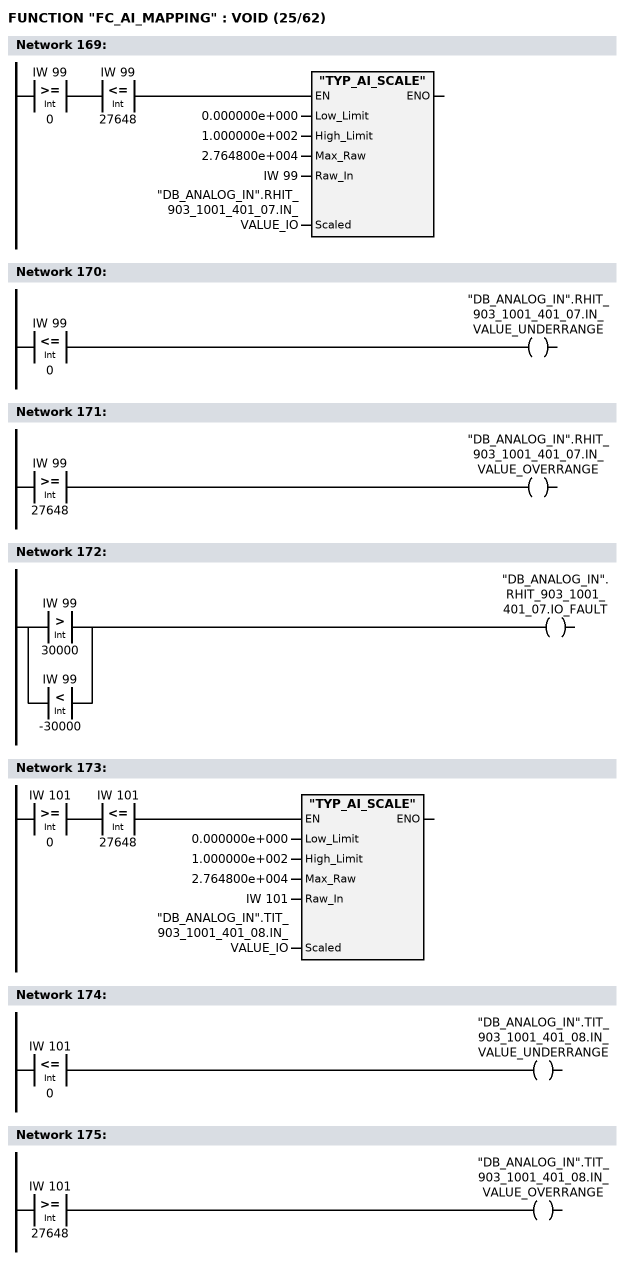

      A(    ;
      L     IW      99;
      L     0;
      >=I   ;
      )     ;
      A(    ;
      L     IW      99;

      L     27648;
      <=I   ;
      )     ;
      JNB   _02b;
      CALL "TYP_AI_SCALE" (
           Low_Limit                := 0.000000e+000,
           High_Limit               := 1.000000e+002,
           Max_Raw                  := 2.764800e+004,
           Raw_In                   := IW      99,
           Scaled                   := "DB_ANALOG_IN".RHIT_903_1001_401_07.IN_VALUE_IO);
_02b: NOP   0;
NETWORK
TITLE =

      L     IW      99;
      L     0;
      <=I   ;
      =     "DB_ANALOG_IN".RHIT_903_1001_401_07.IN_VALUE_UNDERRANGE;
NETWORK
TITLE =

      L     IW      99;
      L     27648;
      >=I   ;
      =     "DB_ANALOG_IN".RHIT_903_1001_401_07.IN_VALUE_OVERRANGE;
NETWORK
TITLE =

      O(    ;
      L     IW      99;
      L     30000;
      >I    ;
      )     ;
      O(    ;
      L     IW      99;
      L     -30000;
      <I    ;
      )     ;
      =     "DB_ANALOG_IN".RHIT_903_1001_401_07.IO_FAULT;

NETWORK
TITLE =

      A(    ;
      L     IW      101;
      L     0;
      >=I   ;
      )     ;
      A(    ;
      L     IW      101;

      L     27648;
      <=I   ;
      )     ;
      JNB   _02c;
      CALL "TYP_AI_SCALE" (
           Low_Limit                := 0.000000e+000,
           High_Limit               := 1.000000e+002,
           Max_Raw                  := 2.764800e+004,
           Raw_In                   := IW      101,
           Scaled                   := "DB_ANALOG_IN".TIT_903_1001_401_08.IN_VALUE_IO);
_02c: NOP   0;
NETWORK
TITLE =

      L     IW      101;
      L     0;
      <=I   ;
      =     "DB_ANALOG_IN".TIT_903_1001_401_08.IN_VALUE_UNDERRANGE;
NETWORK
TITLE =

      L     IW      101;
      L     27648;
      >=I   ;
      =     "DB_ANALOG_IN".TIT_903_1001_401_08.IN_VALUE_OVERRANGE;
NETWORK
TITLE =
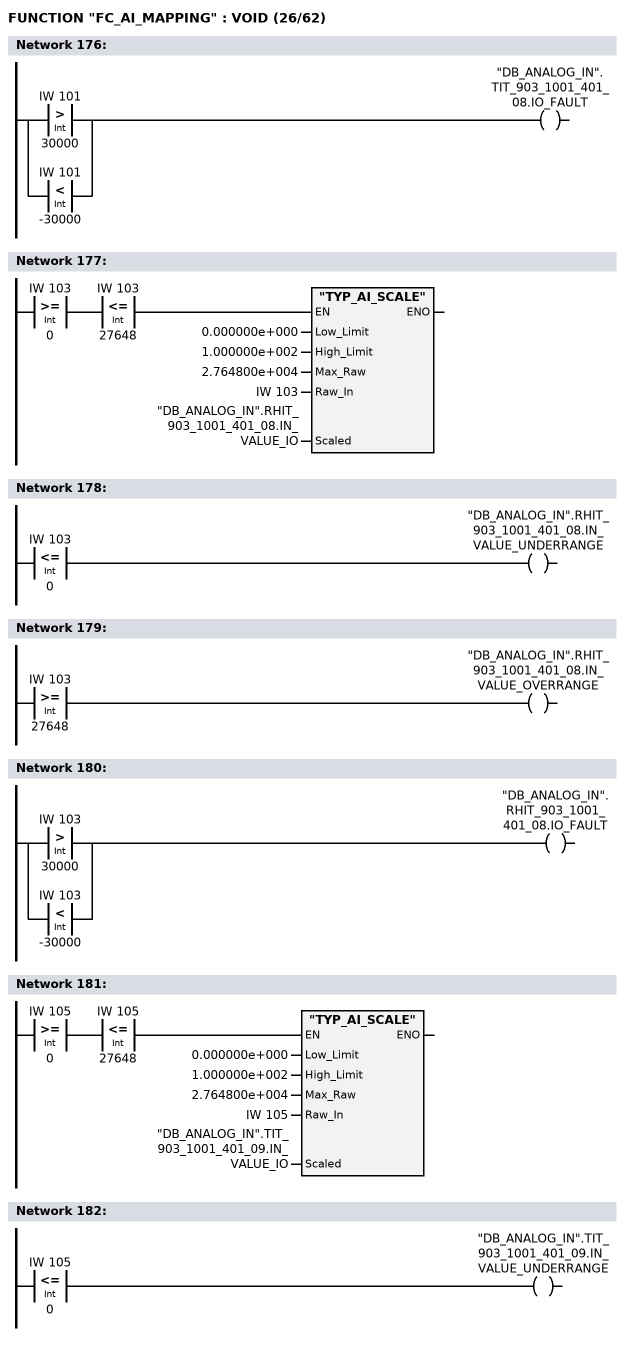

      O(    ;
      L     IW      101;
      L     30000;
      >I    ;
      )     ;
      O(    ;
      L     IW      101;
      L     -30000;
      <I    ;
      )     ;
      =     "DB_ANALOG_IN".TIT_903_1001_401_08.IO_FAULT;

NETWORK
TITLE =

      A(    ;
      L     IW      103;
      L     0;
      >=I   ;
      )     ;
      A(    ;
      L     IW      103;

      L     27648;
      <=I   ;
      )     ;
      JNB   _02d;
      CALL "TYP_AI_SCALE" (
           Low_Limit                := 0.000000e+000,
           High_Limit               := 1.000000e+002,
           Max_Raw                  := 2.764800e+004,
           Raw_In                   := IW      103,
           Scaled                   := "DB_ANALOG_IN".RHIT_903_1001_401_08.IN_VALUE_IO);
_02d: NOP   0;
NETWORK
TITLE =

      L     IW      103;
      L     0;
      <=I   ;
      =     "DB_ANALOG_IN".RHIT_903_1001_401_08.IN_VALUE_UNDERRANGE;
NETWORK
TITLE =

      L     IW      103;
      L     27648;
      >=I   ;
      =     "DB_ANALOG_IN".RHIT_903_1001_401_08.IN_VALUE_OVERRANGE;
NETWORK
TITLE =

      O(    ;
      L     IW      103;
      L     30000;
      >I    ;
      )     ;
      O(    ;
      L     IW      103;
      L     -30000;
      <I    ;
      )     ;
      =     "DB_ANALOG_IN".RHIT_903_1001_401_08.IO_FAULT;

NETWORK
TITLE =

      A(    ;
      L     IW      105;
      L     0;
      >=I   ;
      )     ;
      A(    ;
      L     IW      105;

      L     27648;
      <=I   ;
      )     ;
      JNB   _02e;
      CALL "TYP_AI_SCALE" (
           Low_Limit                := 0.000000e+000,
           High_Limit               := 1.000000e+002,
           Max_Raw                  := 2.764800e+004,
           Raw_In                   := IW      105,
           Scaled                   := "DB_ANALOG_IN".TIT_903_1001_401_09.IN_VALUE_IO);
_02e: NOP   0;
NETWORK
TITLE =

      L     IW      105;
      L     0;
      <=I   ;
      =     "DB_ANALOG_IN".TIT_903_1001_401_09.IN_VALUE_UNDERRANGE;
NETWORK
TITLE =
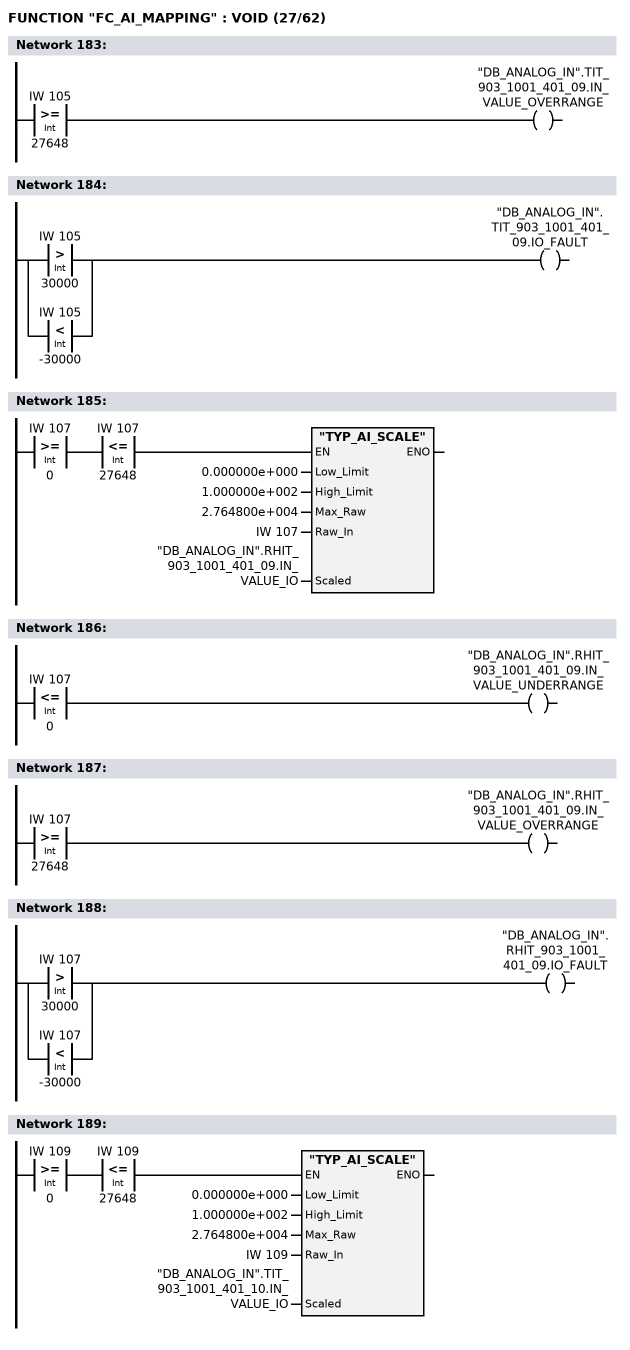

      L     IW      105;
      L     27648;
      >=I   ;
      =     "DB_ANALOG_IN".TIT_903_1001_401_09.IN_VALUE_OVERRANGE;
NETWORK
TITLE =

      O(    ;
      L     IW      105;
      L     30000;
      >I    ;
      )     ;
      O(    ;
      L     IW      105;
      L     -30000;
      <I    ;
      )     ;
      =     "DB_ANALOG_IN".TIT_903_1001_401_09.IO_FAULT;

NETWORK
TITLE =

      A(    ;
      L     IW      107;
      L     0;
      >=I   ;
      )     ;
      A(    ;
      L     IW      107;

      L     27648;
      <=I   ;
      )     ;
      JNB   _02f;
      CALL "TYP_AI_SCALE" (
           Low_Limit                := 0.000000e+000,
           High_Limit               := 1.000000e+002,
           Max_Raw                  := 2.764800e+004,
           Raw_In                   := IW      107,
           Scaled                   := "DB_ANALOG_IN".RHIT_903_1001_401_09.IN_VALUE_IO);
_02f: NOP   0;
NETWORK
TITLE =

      L     IW      107;
      L     0;
      <=I   ;
      =     "DB_ANALOG_IN".RHIT_903_1001_401_09.IN_VALUE_UNDERRANGE;
NETWORK
TITLE =

      L     IW      107;
      L     27648;
      >=I   ;
      =     "DB_ANALOG_IN".RHIT_903_1001_401_09.IN_VALUE_OVERRANGE;
NETWORK
TITLE =

      O(    ;
      L     IW      107;
      L     30000;
      >I    ;
      )     ;
      O(    ;
      L     IW      107;
      L     -30000;
      <I    ;
      )     ;
      =     "DB_ANALOG_IN".RHIT_903_1001_401_09.IO_FAULT;

NETWORK
TITLE =

      A(    ;
      L     IW      109;
      L     0;
      >=I   ;
      )     ;
      A(    ;
      L     IW      109;

      L     27648;
      <=I   ;
      )     ;
      JNB   _030;
      CALL "TYP_AI_SCALE" (
           Low_Limit                := 0.000000e+000,
           High_Limit               := 1.000000e+002,
           Max_Raw                  := 2.764800e+004,
           Raw_In                   := IW      109,
           Scaled                   := "DB_ANALOG_IN".TIT_903_1001_401_10.IN_VALUE_IO);
_030: NOP   0;
NETWORK
TITLE =
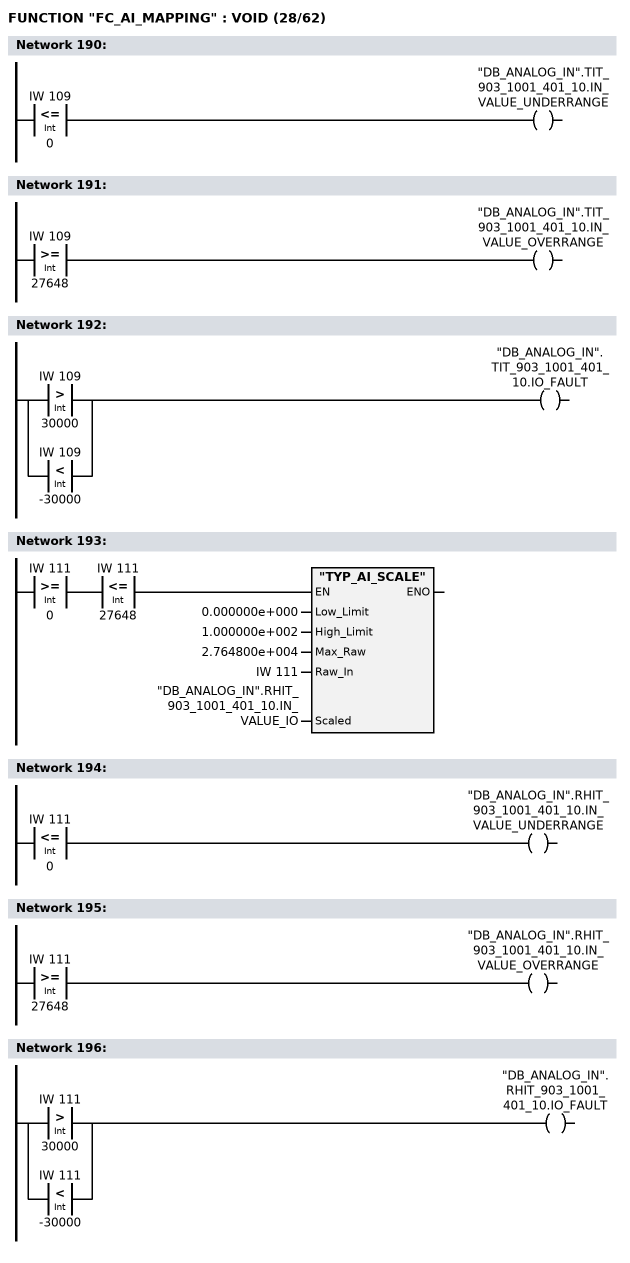

      L     IW      109;
      L     0;
      <=I   ;
      =     "DB_ANALOG_IN".TIT_903_1001_401_10.IN_VALUE_UNDERRANGE;
NETWORK
TITLE =

      L     IW      109;
      L     27648;
      >=I   ;
      =     "DB_ANALOG_IN".TIT_903_1001_401_10.IN_VALUE_OVERRANGE;
NETWORK
TITLE =

      O(    ;
      L     IW      109;
      L     30000;
      >I    ;
      )     ;
      O(    ;
      L     IW      109;
      L     -30000;
      <I    ;
      )     ;
      =     "DB_ANALOG_IN".TIT_903_1001_401_10.IO_FAULT;

NETWORK
TITLE =

      A(    ;
      L     IW      111;
      L     0;
      >=I   ;
      )     ;
      A(    ;
      L     IW      111;

      L     27648;
      <=I   ;
      )     ;
      JNB   _031;
      CALL "TYP_AI_SCALE" (
           Low_Limit                := 0.000000e+000,
           High_Limit               := 1.000000e+002,
           Max_Raw                  := 2.764800e+004,
           Raw_In                   := IW      111,
           Scaled                   := "DB_ANALOG_IN".RHIT_903_1001_401_10.IN_VALUE_IO);
_031: NOP   0;
NETWORK
TITLE =

      L     IW      111;
      L     0;
      <=I   ;
      =     "DB_ANALOG_IN".RHIT_903_1001_401_10.IN_VALUE_UNDERRANGE;
NETWORK
TITLE =

      L     IW      111;
      L     27648;
      >=I   ;
      =     "DB_ANALOG_IN".RHIT_903_1001_401_10.IN_VALUE_OVERRANGE;
NETWORK
TITLE =

      O(    ;
      L     IW      111;
      L     30000;
      >I    ;
      )     ;
      O(    ;
      L     IW      111;
      L     -30000;
      <I    ;
      )     ;
      =     "DB_ANALOG_IN".RHIT_903_1001_401_10.IO_FAULT;

NETWORK
TITLE =
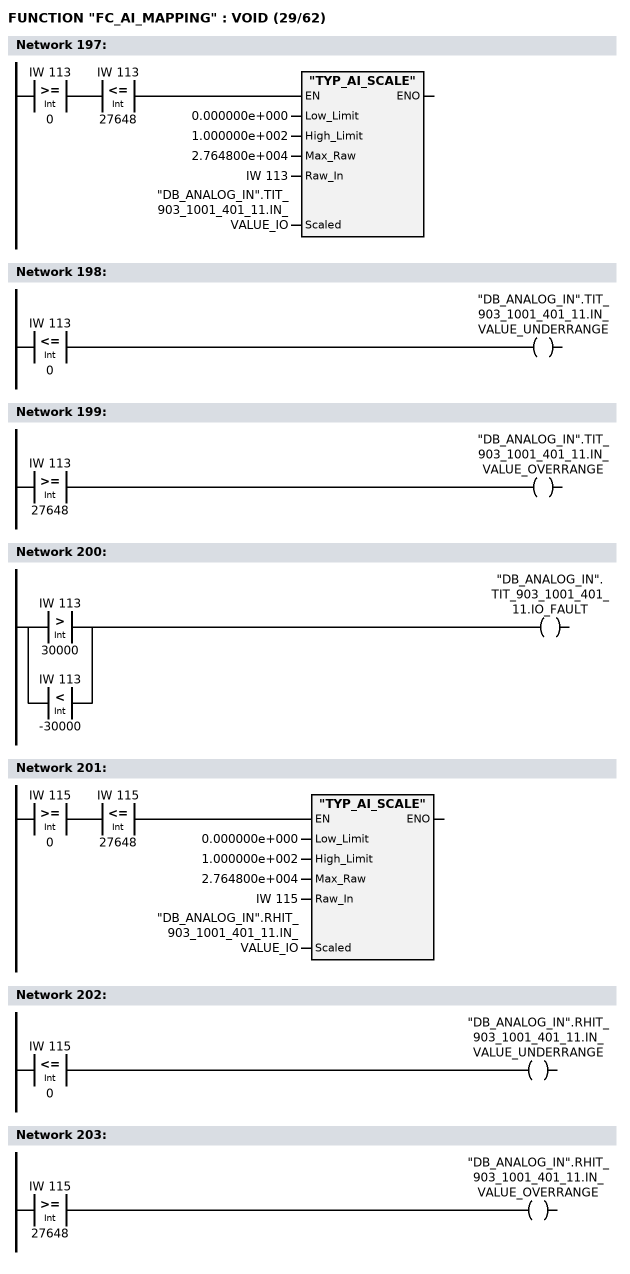

      A(    ;
      L     IW      113;
      L     0;
      >=I   ;
      )     ;
      A(    ;
      L     IW      113;

      L     27648;
      <=I   ;
      )     ;
      JNB   _032;
      CALL "TYP_AI_SCALE" (
           Low_Limit                := 0.000000e+000,
           High_Limit               := 1.000000e+002,
           Max_Raw                  := 2.764800e+004,
           Raw_In                   := IW      113,
           Scaled                   := "DB_ANALOG_IN".TIT_903_1001_401_11.IN_VALUE_IO);
_032: NOP   0;
NETWORK
TITLE =

      L     IW      113;
      L     0;
      <=I   ;
      =     "DB_ANALOG_IN".TIT_903_1001_401_11.IN_VALUE_UNDERRANGE;
NETWORK
TITLE =

      L     IW      113;
      L     27648;
      >=I   ;
      =     "DB_ANALOG_IN".TIT_903_1001_401_11.IN_VALUE_OVERRANGE;
NETWORK
TITLE =

      O(    ;
      L     IW      113;
      L     30000;
      >I    ;
      )     ;
      O(    ;
      L     IW      113;
      L     -30000;
      <I    ;
      )     ;
      =     "DB_ANALOG_IN".TIT_903_1001_401_11.IO_FAULT;

NETWORK
TITLE =

      A(    ;
      L     IW      115;
      L     0;
      >=I   ;
      )     ;
      A(    ;
      L     IW      115;

      L     27648;
      <=I   ;
      )     ;
      JNB   _033;
      CALL "TYP_AI_SCALE" (
           Low_Limit                := 0.000000e+000,
           High_Limit               := 1.000000e+002,
           Max_Raw                  := 2.764800e+004,
           Raw_In                   := IW      115,
           Scaled                   := "DB_ANALOG_IN".RHIT_903_1001_401_11.IN_VALUE_IO);
_033: NOP   0;
NETWORK
TITLE =

      L     IW      115;
      L     0;
      <=I   ;
      =     "DB_ANALOG_IN".RHIT_903_1001_401_11.IN_VALUE_UNDERRANGE;
NETWORK
TITLE =

      L     IW      115;
      L     27648;
      >=I   ;
      =     "DB_ANALOG_IN".RHIT_903_1001_401_11.IN_VALUE_OVERRANGE;
NETWORK
TITLE =
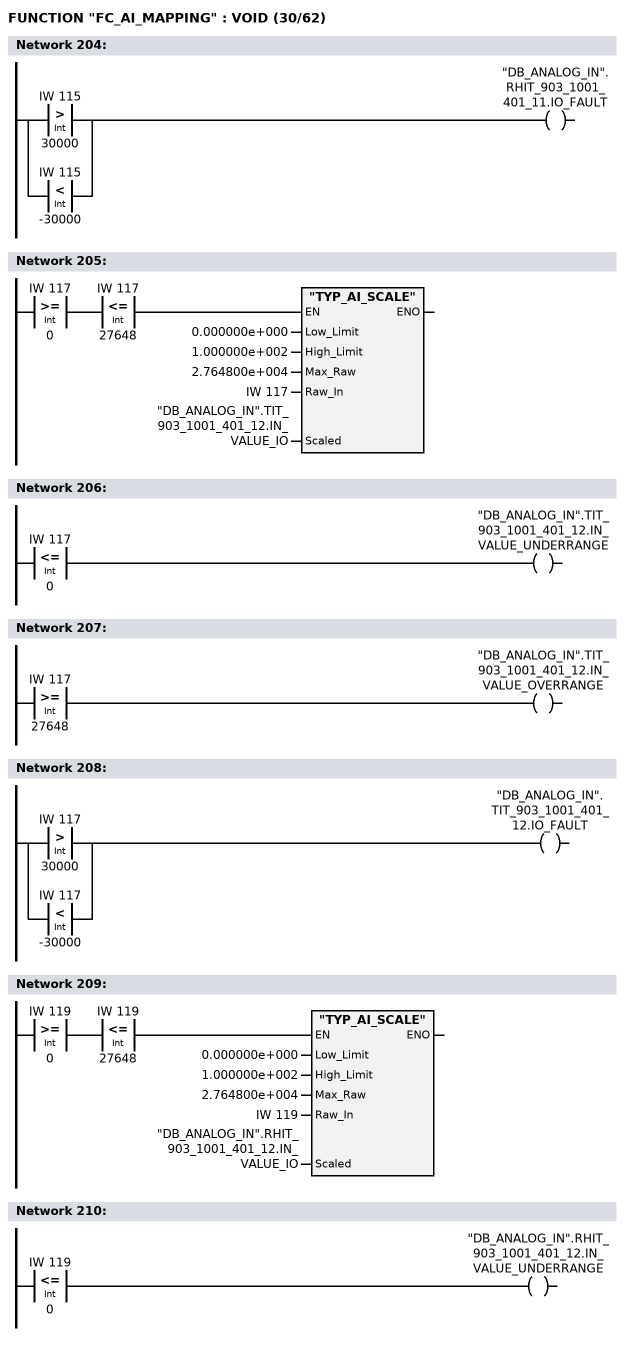

      O(    ;
      L     IW      115;
      L     30000;
      >I    ;
      )     ;
      O(    ;
      L     IW      115;
      L     -30000;
      <I    ;
      )     ;
      =     "DB_ANALOG_IN".RHIT_903_1001_401_11.IO_FAULT;

NETWORK
TITLE =

      A(    ;
      L     IW      117;
      L     0;
      >=I   ;
      )     ;
      A(    ;
      L     IW      117;

      L     27648;
      <=I   ;
      )     ;
      JNB   _034;
      CALL "TYP_AI_SCALE" (
           Low_Limit                := 0.000000e+000,
           High_Limit               := 1.000000e+002,
           Max_Raw                  := 2.764800e+004,
           Raw_In                   := IW      117,
           Scaled                   := "DB_ANALOG_IN".TIT_903_1001_401_12.IN_VALUE_IO);
_034: NOP   0;
NETWORK
TITLE =

      L     IW      117;
      L     0;
      <=I   ;
      =     "DB_ANALOG_IN".TIT_903_1001_401_12.IN_VALUE_UNDERRANGE;
NETWORK
TITLE =

      L     IW      117;
      L     27648;
      >=I   ;
      =     "DB_ANALOG_IN".TIT_903_1001_401_12.IN_VALUE_OVERRANGE;
NETWORK
TITLE =

      O(    ;
      L     IW      117;
      L     30000;
      >I    ;
      )     ;
      O(    ;
      L     IW      117;
      L     -30000;
      <I    ;
      )     ;
      =     "DB_ANALOG_IN".TIT_903_1001_401_12.IO_FAULT;

NETWORK
TITLE =

      A(    ;
      L     IW      119;
      L     0;
      >=I   ;
      )     ;
      A(    ;
      L     IW      119;

      L     27648;
      <=I   ;
      )     ;
      JNB   _035;
      CALL "TYP_AI_SCALE" (
           Low_Limit                := 0.000000e+000,
           High_Limit               := 1.000000e+002,
           Max_Raw                  := 2.764800e+004,
           Raw_In                   := IW      119,
           Scaled                   := "DB_ANALOG_IN".RHIT_903_1001_401_12.IN_VALUE_IO);
_035: NOP   0;
NETWORK
TITLE =

      L     IW      119;
      L     0;
      <=I   ;
      =     "DB_ANALOG_IN".RHIT_903_1001_401_12.IN_VALUE_UNDERRANGE;
NETWORK
TITLE =
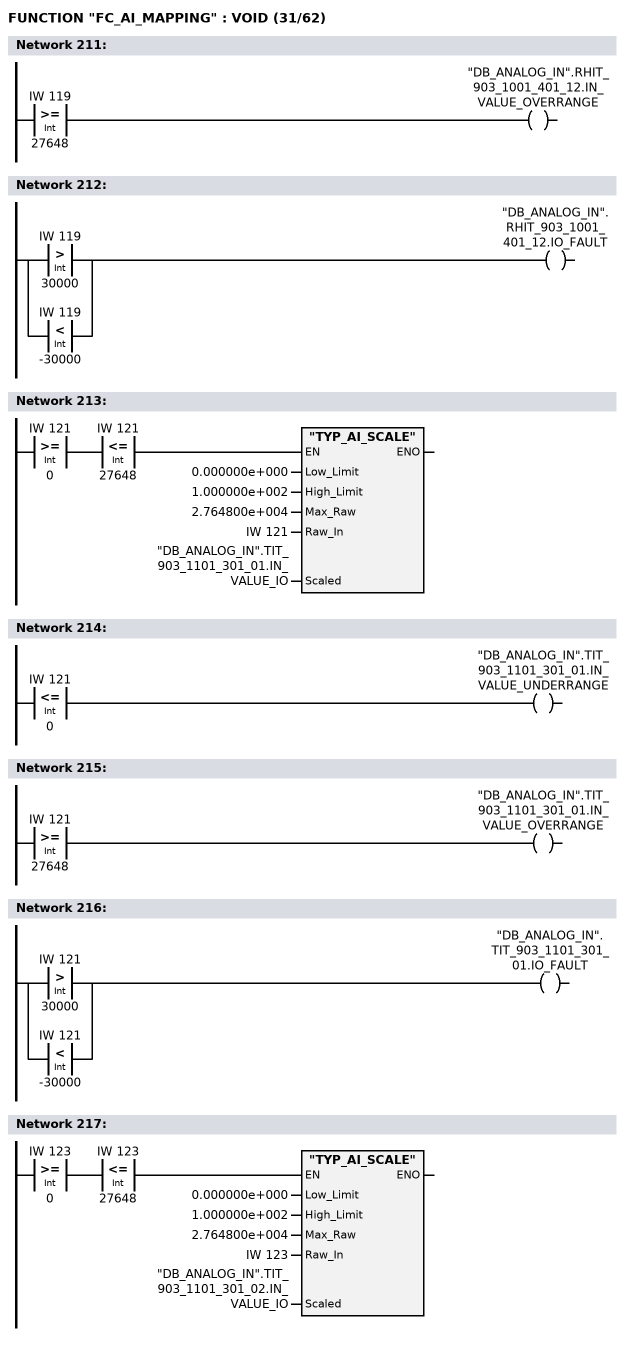

      L     IW      119;
      L     27648;
      >=I   ;
      =     "DB_ANALOG_IN".RHIT_903_1001_401_12.IN_VALUE_OVERRANGE;
NETWORK
TITLE =

      O(    ;
      L     IW      119;
      L     30000;
      >I    ;
      )     ;
      O(    ;
      L     IW      119;
      L     -30000;
      <I    ;
      )     ;
      =     "DB_ANALOG_IN".RHIT_903_1001_401_12.IO_FAULT;

NETWORK
TITLE =

      A(    ;
      L     IW      121;
      L     0;
      >=I   ;
      )     ;
      A(    ;
      L     IW      121;

      L     27648;
      <=I   ;
      )     ;
      JNB   _036;
      CALL "TYP_AI_SCALE" (
           Low_Limit                := 0.000000e+000,
           High_Limit               := 1.000000e+002,
           Max_Raw                  := 2.764800e+004,
           Raw_In                   := IW      121,
           Scaled                   := "DB_ANALOG_IN".TIT_903_1101_301_01.IN_VALUE_IO);
_036: NOP   0;
NETWORK
TITLE =

      L     IW      121;
      L     0;
      <=I   ;
      =     "DB_ANALOG_IN".TIT_903_1101_301_01.IN_VALUE_UNDERRANGE;
NETWORK
TITLE =

      L     IW      121;
      L     27648;
      >=I   ;
      =     "DB_ANALOG_IN".TIT_903_1101_301_01.IN_VALUE_OVERRANGE;
NETWORK
TITLE =

      O(    ;
      L     IW      121;
      L     30000;
      >I    ;
      )     ;
      O(    ;
      L     IW      121;
      L     -30000;
      <I    ;
      )     ;
      =     "DB_ANALOG_IN".TIT_903_1101_301_01.IO_FAULT;

NETWORK
TITLE =

      A(    ;
      L     IW      123;
      L     0;
      >=I   ;
      )     ;
      A(    ;
      L     IW      123;

      L     27648;
      <=I   ;
      )     ;
      JNB   _037;
      CALL "TYP_AI_SCALE" (
           Low_Limit                := 0.000000e+000,
           High_Limit               := 1.000000e+002,
           Max_Raw                  := 2.764800e+004,
           Raw_In                   := IW      123,
           Scaled                   := "DB_ANALOG_IN".TIT_903_1101_301_02.IN_VALUE_IO);
_037: NOP   0;
NETWORK
TITLE =
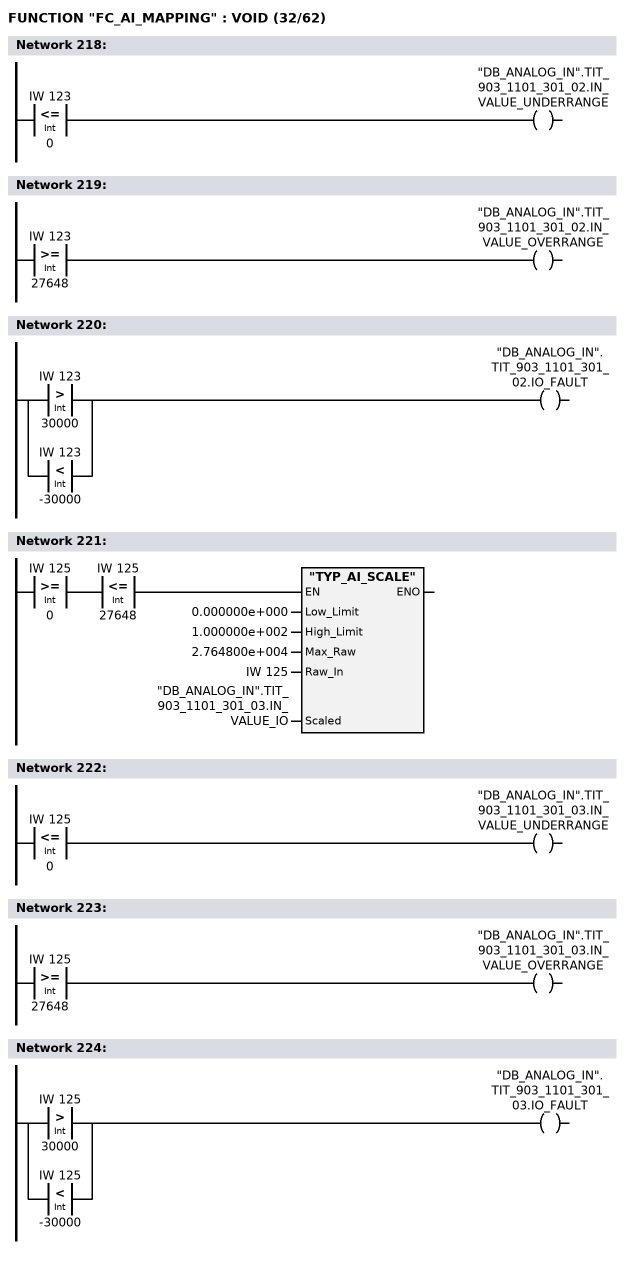

      L     IW      123;
      L     0;
      <=I   ;
      =     "DB_ANALOG_IN".TIT_903_1101_301_02.IN_VALUE_UNDERRANGE;
NETWORK
TITLE =

      L     IW      123;
      L     27648;
      >=I   ;
      =     "DB_ANALOG_IN".TIT_903_1101_301_02.IN_VALUE_OVERRANGE;
NETWORK
TITLE =

      O(    ;
      L     IW      123;
      L     30000;
      >I    ;
      )     ;
      O(    ;
      L     IW      123;
      L     -30000;
      <I    ;
      )     ;
      =     "DB_ANALOG_IN".TIT_903_1101_301_02.IO_FAULT;

NETWORK
TITLE =

      A(    ;
      L     IW      125;
      L     0;
      >=I   ;
      )     ;
      A(    ;
      L     IW      125;

      L     27648;
      <=I   ;
      )     ;
      JNB   _038;
      CALL "TYP_AI_SCALE" (
           Low_Limit                := 0.000000e+000,
           High_Limit               := 1.000000e+002,
           Max_Raw                  := 2.764800e+004,
           Raw_In                   := IW      125,
           Scaled                   := "DB_ANALOG_IN".TIT_903_1101_301_03.IN_VALUE_IO);
_038: NOP   0;
NETWORK
TITLE =

      L     IW      125;
      L     0;
      <=I   ;
      =     "DB_ANALOG_IN".TIT_903_1101_301_03.IN_VALUE_UNDERRANGE;
NETWORK
TITLE =

      L     IW      125;
      L     27648;
      >=I   ;
      =     "DB_ANALOG_IN".TIT_903_1101_301_03.IN_VALUE_OVERRANGE;
NETWORK
TITLE =

      O(    ;
      L     IW      125;
      L     30000;
      >I    ;
      )     ;
      O(    ;
      L     IW      125;
      L     -30000;
      <I    ;
      )     ;
      =     "DB_ANALOG_IN".TIT_903_1101_301_03.IO_FAULT;

NETWORK
TITLE =
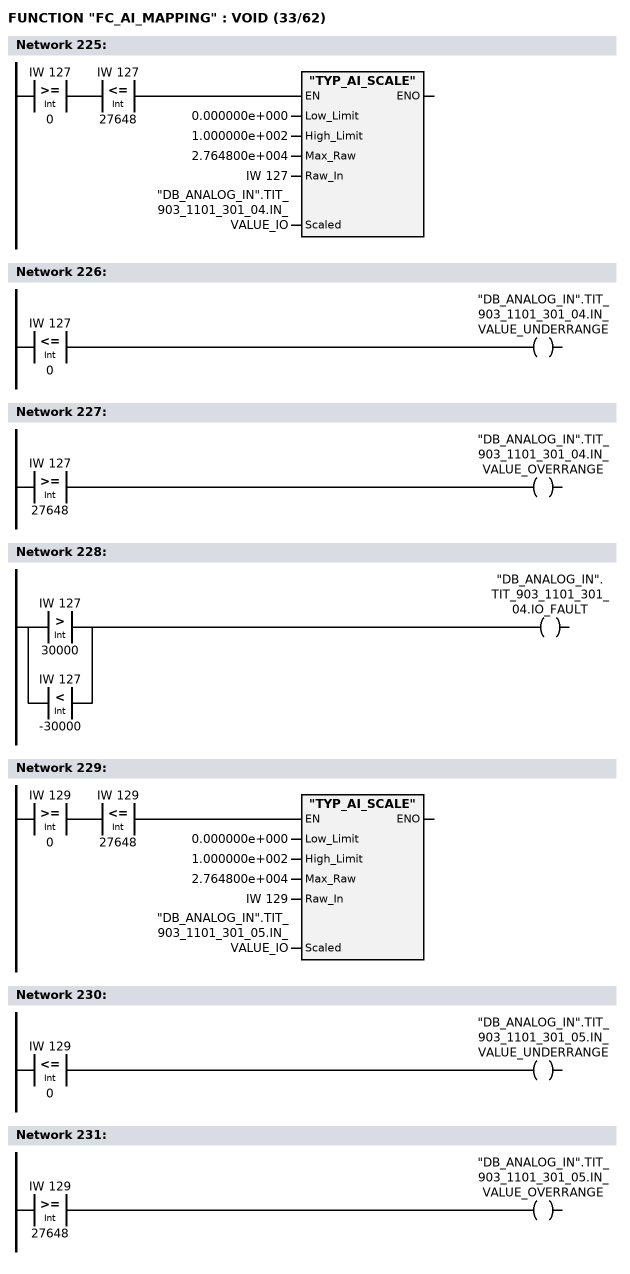

      A(    ;
      L     IW      127;
      L     0;
      >=I   ;
      )     ;
      A(    ;
      L     IW      127;

      L     27648;
      <=I   ;
      )     ;
      JNB   _039;
      CALL "TYP_AI_SCALE" (
           Low_Limit                := 0.000000e+000,
           High_Limit               := 1.000000e+002,
           Max_Raw                  := 2.764800e+004,
           Raw_In                   := IW      127,
           Scaled                   := "DB_ANALOG_IN".TIT_903_1101_301_04.IN_VALUE_IO);
_039: NOP   0;
NETWORK
TITLE =

      L     IW      127;
      L     0;
      <=I   ;
      =     "DB_ANALOG_IN".TIT_903_1101_301_04.IN_VALUE_UNDERRANGE;
NETWORK
TITLE =

      L     IW      127;
      L     27648;
      >=I   ;
      =     "DB_ANALOG_IN".TIT_903_1101_301_04.IN_VALUE_OVERRANGE;
NETWORK
TITLE =

      O(    ;
      L     IW      127;
      L     30000;
      >I    ;
      )     ;
      O(    ;
      L     IW      127;
      L     -30000;
      <I    ;
      )     ;
      =     "DB_ANALOG_IN".TIT_903_1101_301_04.IO_FAULT;

NETWORK
TITLE =

      A(    ;
      L     IW      129;
      L     0;
      >=I   ;
      )     ;
      A(    ;
      L     IW      129;

      L     27648;
      <=I   ;
      )     ;
      JNB   _03a;
      CALL "TYP_AI_SCALE" (
           Low_Limit                := 0.000000e+000,
           High_Limit               := 1.000000e+002,
           Max_Raw                  := 2.764800e+004,
           Raw_In                   := IW      129,
           Scaled                   := "DB_ANALOG_IN".TIT_903_1101_301_05.IN_VALUE_IO);
_03a: NOP   0;
NETWORK
TITLE =

      L     IW      129;
      L     0;
      <=I   ;
      =     "DB_ANALOG_IN".TIT_903_1101_301_05.IN_VALUE_UNDERRANGE;
NETWORK
TITLE =

      L     IW      129;
      L     27648;
      >=I   ;
      =     "DB_ANALOG_IN".TIT_903_1101_301_05.IN_VALUE_OVERRANGE;
NETWORK
TITLE =
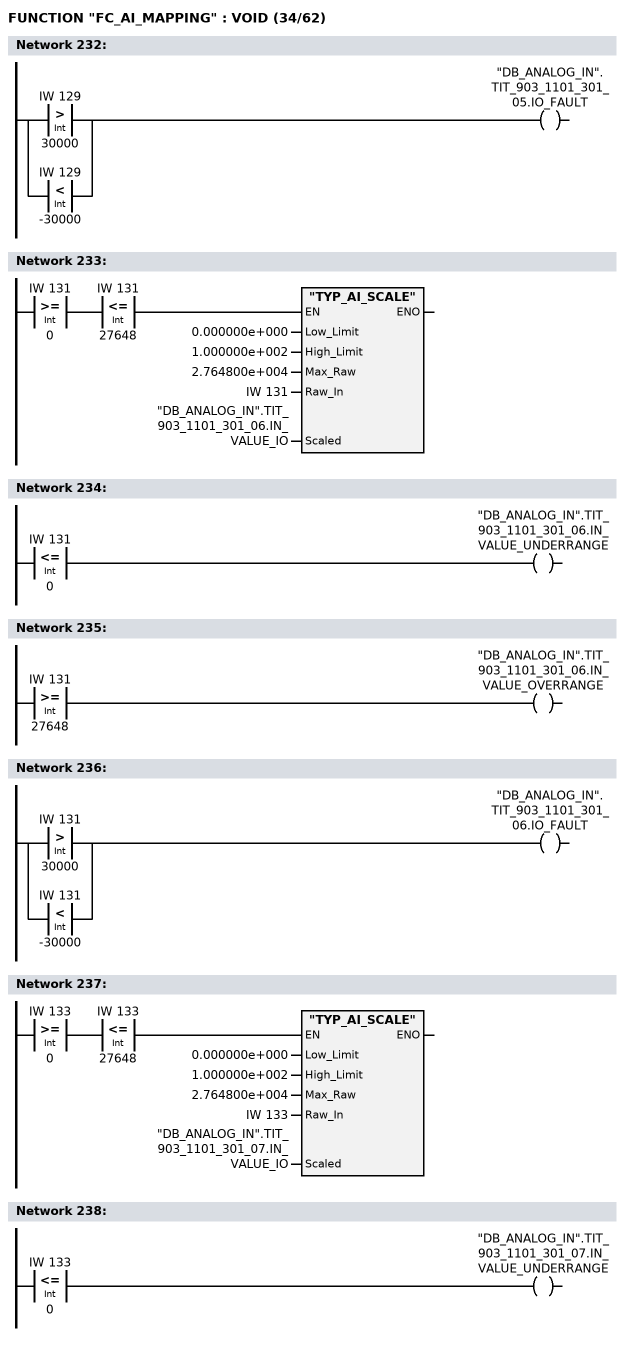

      O(    ;
      L     IW      129;
      L     30000;
      >I    ;
      )     ;
      O(    ;
      L     IW      129;
      L     -30000;
      <I    ;
      )     ;
      =     "DB_ANALOG_IN".TIT_903_1101_301_05.IO_FAULT;

NETWORK
TITLE =

      A(    ;
      L     IW      131;
      L     0;
      >=I   ;
      )     ;
      A(    ;
      L     IW      131;

      L     27648;
      <=I   ;
      )     ;
      JNB   _03b;
      CALL "TYP_AI_SCALE" (
           Low_Limit                := 0.000000e+000,
           High_Limit               := 1.000000e+002,
           Max_Raw                  := 2.764800e+004,
           Raw_In                   := IW      131,
           Scaled                   := "DB_ANALOG_IN".TIT_903_1101_301_06.IN_VALUE_IO);
_03b: NOP   0;
NETWORK
TITLE =

      L     IW      131;
      L     0;
      <=I   ;
      =     "DB_ANALOG_IN".TIT_903_1101_301_06.IN_VALUE_UNDERRANGE;
NETWORK
TITLE =

      L     IW      131;
      L     27648;
      >=I   ;
      =     "DB_ANALOG_IN".TIT_903_1101_301_06.IN_VALUE_OVERRANGE;
NETWORK
TITLE =

      O(    ;
      L     IW      131;
      L     30000;
      >I    ;
      )     ;
      O(    ;
      L     IW      131;
      L     -30000;
      <I    ;
      )     ;
      =     "DB_ANALOG_IN".TIT_903_1101_301_06.IO_FAULT;

NETWORK
TITLE =

      A(    ;
      L     IW      133;
      L     0;
      >=I   ;
      )     ;
      A(    ;
      L     IW      133;

      L     27648;
      <=I   ;
      )     ;
      JNB   _03c;
      CALL "TYP_AI_SCALE" (
           Low_Limit                := 0.000000e+000,
           High_Limit               := 1.000000e+002,
           Max_Raw                  := 2.764800e+004,
           Raw_In                   := IW      133,
           Scaled                   := "DB_ANALOG_IN".TIT_903_1101_301_07.IN_VALUE_IO);
_03c: NOP   0;
NETWORK
TITLE =

      L     IW      133;
      L     0;
      <=I   ;
      =     "DB_ANALOG_IN".TIT_903_1101_301_07.IN_VALUE_UNDERRANGE;
NETWORK
TITLE =
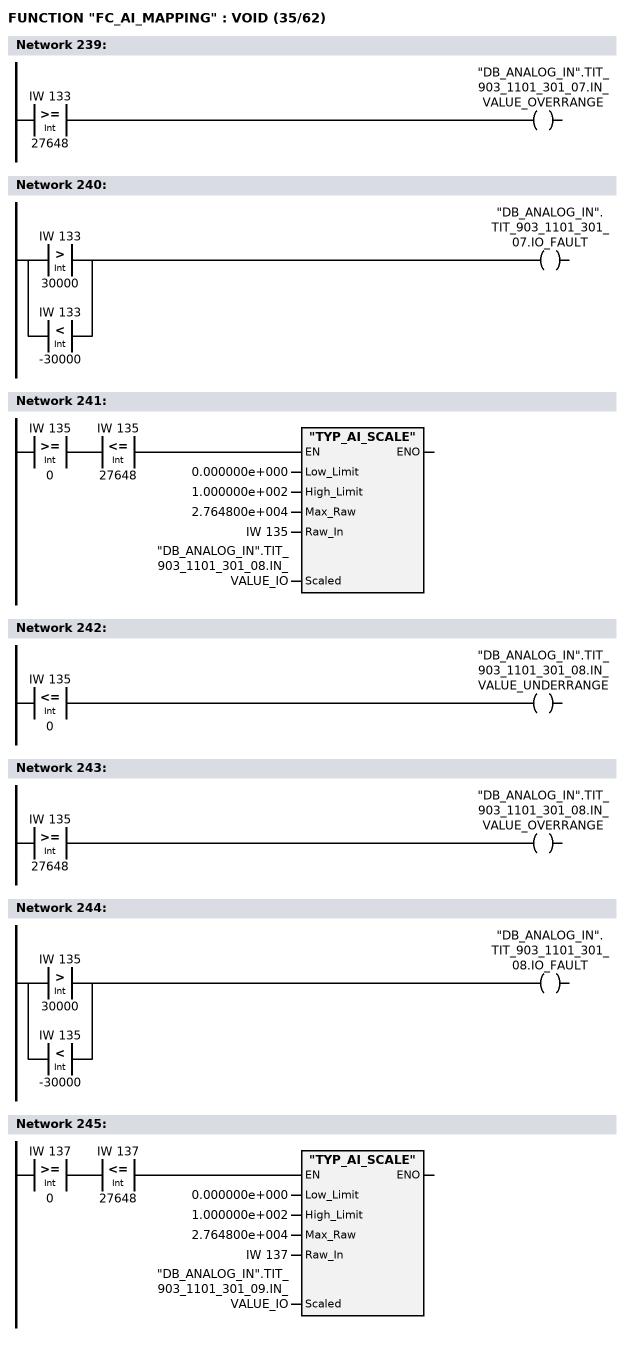

      L     IW      133;
      L     27648;
      >=I   ;
      =     "DB_ANALOG_IN".TIT_903_1101_301_07.IN_VALUE_OVERRANGE;
NETWORK
TITLE =

      O(    ;
      L     IW      133;
      L     30000;
      >I    ;
      )     ;
      O(    ;
      L     IW      133;
      L     -30000;
      <I    ;
      )     ;
      =     "DB_ANALOG_IN".TIT_903_1101_301_07.IO_FAULT;

NETWORK
TITLE =

      A(    ;
      L     IW      135;
      L     0;
      >=I   ;
      )     ;
      A(    ;
      L     IW      135;

      L     27648;
      <=I   ;
      )     ;
      JNB   _03d;
      CALL "TYP_AI_SCALE" (
           Low_Limit                := 0.000000e+000,
           High_Limit               := 1.000000e+002,
           Max_Raw                  := 2.764800e+004,
           Raw_In                   := IW      135,
           Scaled                   := "DB_ANALOG_IN".TIT_903_1101_301_08.IN_VALUE_IO);
_03d: NOP   0;
NETWORK
TITLE =

      L     IW      135;
      L     0;
      <=I   ;
      =     "DB_ANALOG_IN".TIT_903_1101_301_08.IN_VALUE_UNDERRANGE;
NETWORK
TITLE =

      L     IW      135;
      L     27648;
      >=I   ;
      =     "DB_ANALOG_IN".TIT_903_1101_301_08.IN_VALUE_OVERRANGE;
NETWORK
TITLE =

      O(    ;
      L     IW      135;
      L     30000;
      >I    ;
      )     ;
      O(    ;
      L     IW      135;
      L     -30000;
      <I    ;
      )     ;
      =     "DB_ANALOG_IN".TIT_903_1101_301_08.IO_FAULT;

NETWORK
TITLE =

      A(    ;
      L     IW      137;
      L     0;
      >=I   ;
      )     ;
      A(    ;
      L     IW      137;

      L     27648;
      <=I   ;
      )     ;
      JNB   _03e;
      CALL "TYP_AI_SCALE" (
           Low_Limit                := 0.000000e+000,
           High_Limit               := 1.000000e+002,
           Max_Raw                  := 2.764800e+004,
           Raw_In                   := IW      137,
           Scaled                   := "DB_ANALOG_IN".TIT_903_1101_301_09.IN_VALUE_IO);
_03e: NOP   0;
NETWORK
TITLE =
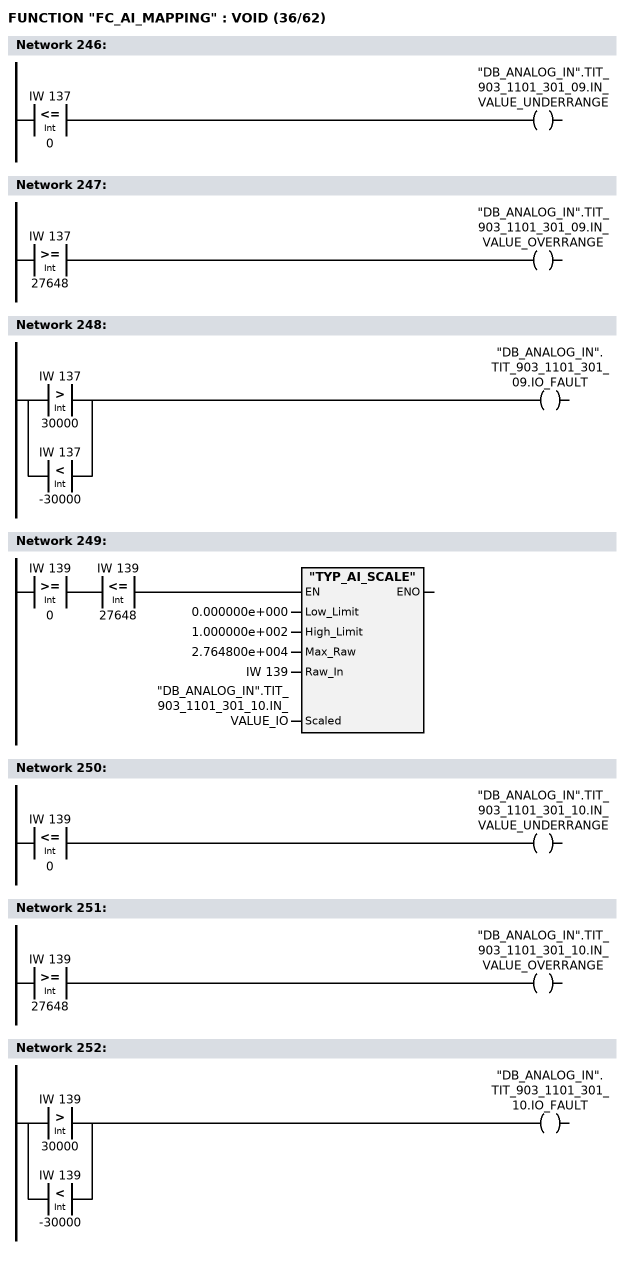

      L     IW      137;
      L     0;
      <=I   ;
      =     "DB_ANALOG_IN".TIT_903_1101_301_09.IN_VALUE_UNDERRANGE;
NETWORK
TITLE =

      L     IW      137;
      L     27648;
      >=I   ;
      =     "DB_ANALOG_IN".TIT_903_1101_301_09.IN_VALUE_OVERRANGE;
NETWORK
TITLE =

      O(    ;
      L     IW      137;
      L     30000;
      >I    ;
      )     ;
      O(    ;
      L     IW      137;
      L     -30000;
      <I    ;
      )     ;
      =     "DB_ANALOG_IN".TIT_903_1101_301_09.IO_FAULT;

NETWORK
TITLE =

      A(    ;
      L     IW      139;
      L     0;
      >=I   ;
      )     ;
      A(    ;
      L     IW      139;

      L     27648;
      <=I   ;
      )     ;
      JNB   _03f;
      CALL "TYP_AI_SCALE" (
           Low_Limit                := 0.000000e+000,
           High_Limit               := 1.000000e+002,
           Max_Raw                  := 2.764800e+004,
           Raw_In                   := IW      139,
           Scaled                   := "DB_ANALOG_IN".TIT_903_1101_301_10.IN_VALUE_IO);
_03f: NOP   0;
NETWORK
TITLE =

      L     IW      139;
      L     0;
      <=I   ;
      =     "DB_ANALOG_IN".TIT_903_1101_301_10.IN_VALUE_UNDERRANGE;
NETWORK
TITLE =

      L     IW      139;
      L     27648;
      >=I   ;
      =     "DB_ANALOG_IN".TIT_903_1101_301_10.IN_VALUE_OVERRANGE;
NETWORK
TITLE =

      O(    ;
      L     IW      139;
      L     30000;
      >I    ;
      )     ;
      O(    ;
      L     IW      139;
      L     -30000;
      <I    ;
      )     ;
      =     "DB_ANALOG_IN".TIT_903_1101_301_10.IO_FAULT;

NETWORK
TITLE =
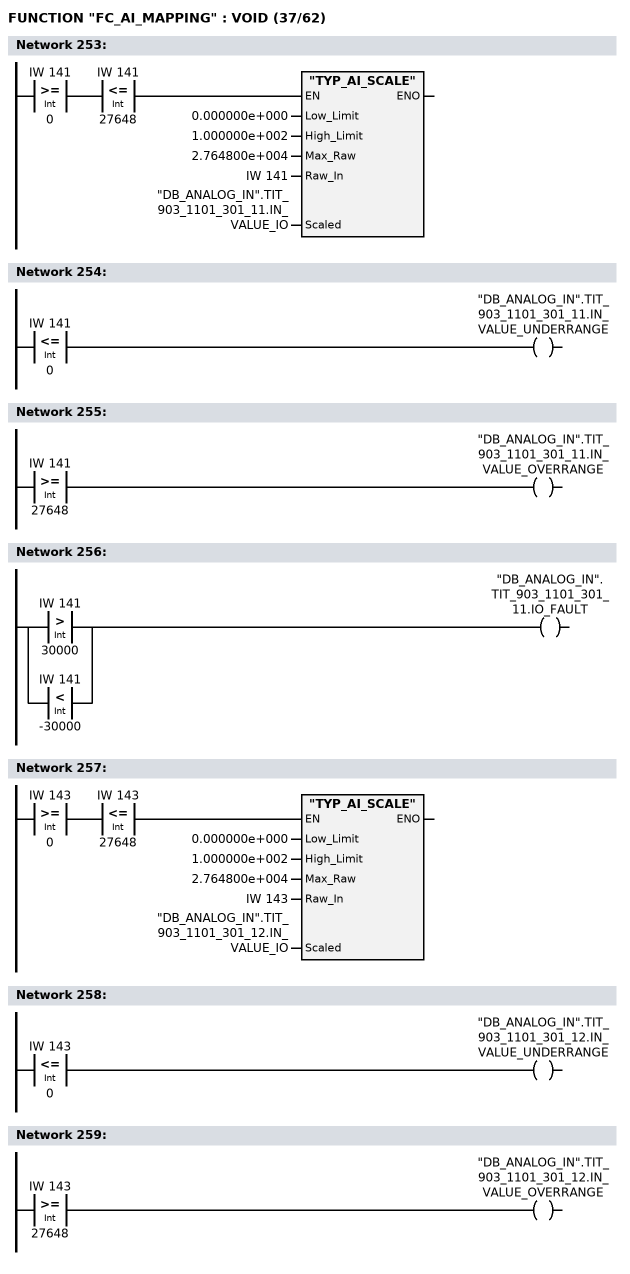

      A(    ;
      L     IW      141;
      L     0;
      >=I   ;
      )     ;
      A(    ;
      L     IW      141;

      L     27648;
      <=I   ;
      )     ;
      JNB   _040;
      CALL "TYP_AI_SCALE" (
           Low_Limit                := 0.000000e+000,
           High_Limit               := 1.000000e+002,
           Max_Raw                  := 2.764800e+004,
           Raw_In                   := IW      141,
           Scaled                   := "DB_ANALOG_IN".TIT_903_1101_301_11.IN_VALUE_IO);
_040: NOP   0;
NETWORK
TITLE =

      L     IW      141;
      L     0;
      <=I   ;
      =     "DB_ANALOG_IN".TIT_903_1101_301_11.IN_VALUE_UNDERRANGE;
NETWORK
TITLE =

      L     IW      141;
      L     27648;
      >=I   ;
      =     "DB_ANALOG_IN".TIT_903_1101_301_11.IN_VALUE_OVERRANGE;
NETWORK
TITLE =

      O(    ;
      L     IW      141;
      L     30000;
      >I    ;
      )     ;
      O(    ;
      L     IW      141;
      L     -30000;
      <I    ;
      )     ;
      =     "DB_ANALOG_IN".TIT_903_1101_301_11.IO_FAULT;

NETWORK
TITLE =

      A(    ;
      L     IW      143;
      L     0;
      >=I   ;
      )     ;
      A(    ;
      L     IW      143;

      L     27648;
      <=I   ;
      )     ;
      JNB   _041;
      CALL "TYP_AI_SCALE" (
           Low_Limit                := 0.000000e+000,
           High_Limit               := 1.000000e+002,
           Max_Raw                  := 2.764800e+004,
           Raw_In                   := IW      143,
           Scaled                   := "DB_ANALOG_IN".TIT_903_1101_301_12.IN_VALUE_IO);
_041: NOP   0;
NETWORK
TITLE =

      L     IW      143;
      L     0;
      <=I   ;
      =     "DB_ANALOG_IN".TIT_903_1101_301_12.IN_VALUE_UNDERRANGE;
NETWORK
TITLE =

      L     IW      143;
      L     27648;
      >=I   ;
      =     "DB_ANALOG_IN".TIT_903_1101_301_12.IN_VALUE_OVERRANGE;
NETWORK
TITLE =
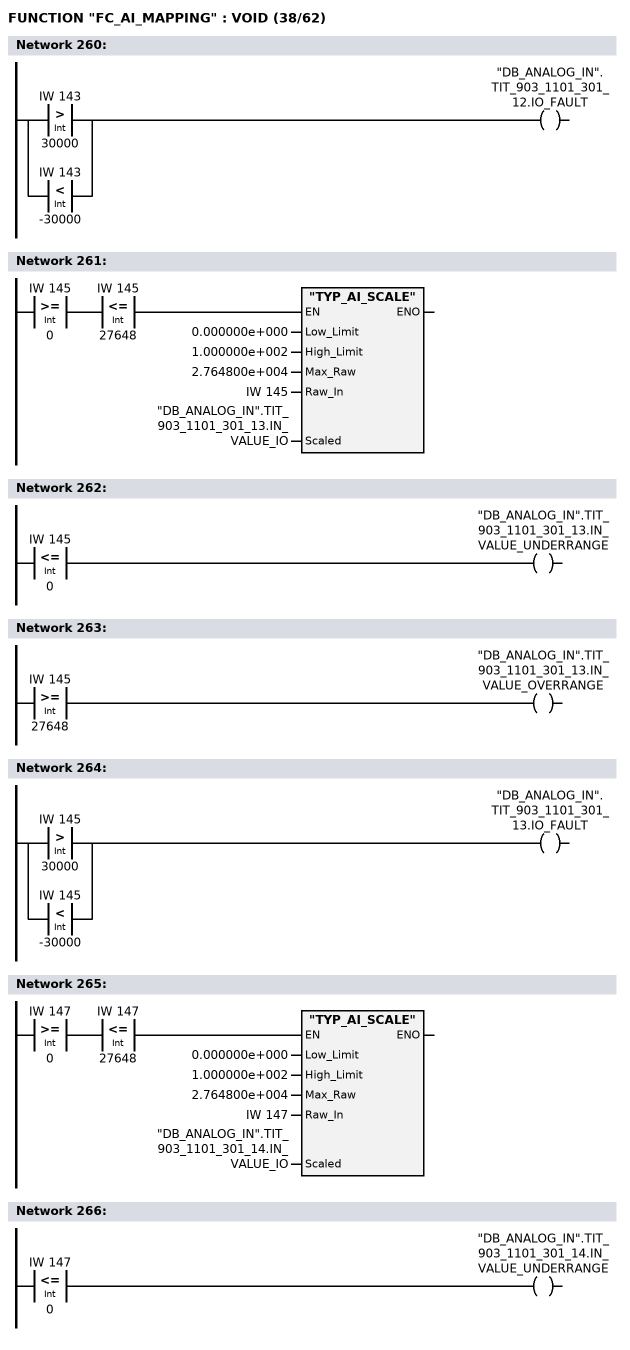

      O(    ;
      L     IW      143;
      L     30000;
      >I    ;
      )     ;
      O(    ;
      L     IW      143;
      L     -30000;
      <I    ;
      )     ;
      =     "DB_ANALOG_IN".TIT_903_1101_301_12.IO_FAULT;

NETWORK
TITLE =

      A(    ;
      L     IW      145;
      L     0;
      >=I   ;
      )     ;
      A(    ;
      L     IW      145;

      L     27648;
      <=I   ;
      )     ;
      JNB   _042;
      CALL "TYP_AI_SCALE" (
           Low_Limit                := 0.000000e+000,
           High_Limit               := 1.000000e+002,
           Max_Raw                  := 2.764800e+004,
           Raw_In                   := IW      145,
           Scaled                   := "DB_ANALOG_IN".TIT_903_1101_301_13.IN_VALUE_IO);
_042: NOP   0;
NETWORK
TITLE =

      L     IW      145;
      L     0;
      <=I   ;
      =     "DB_ANALOG_IN".TIT_903_1101_301_13.IN_VALUE_UNDERRANGE;
NETWORK
TITLE =

      L     IW      145;
      L     27648;
      >=I   ;
      =     "DB_ANALOG_IN".TIT_903_1101_301_13.IN_VALUE_OVERRANGE;
NETWORK
TITLE =

      O(    ;
      L     IW      145;
      L     30000;
      >I    ;
      )     ;
      O(    ;
      L     IW      145;
      L     -30000;
      <I    ;
      )     ;
      =     "DB_ANALOG_IN".TIT_903_1101_301_13.IO_FAULT;

NETWORK
TITLE =

      A(    ;
      L     IW      147;
      L     0;
      >=I   ;
      )     ;
      A(    ;
      L     IW      147;

      L     27648;
      <=I   ;
      )     ;
      JNB   _043;
      CALL "TYP_AI_SCALE" (
           Low_Limit                := 0.000000e+000,
           High_Limit               := 1.000000e+002,
           Max_Raw                  := 2.764800e+004,
           Raw_In                   := IW      147,
           Scaled                   := "DB_ANALOG_IN".TIT_903_1101_301_14.IN_VALUE_IO);
_043: NOP   0;
NETWORK
TITLE =

      L     IW      147;
      L     0;
      <=I   ;
      =     "DB_ANALOG_IN".TIT_903_1101_301_14.IN_VALUE_UNDERRANGE;
NETWORK
TITLE =
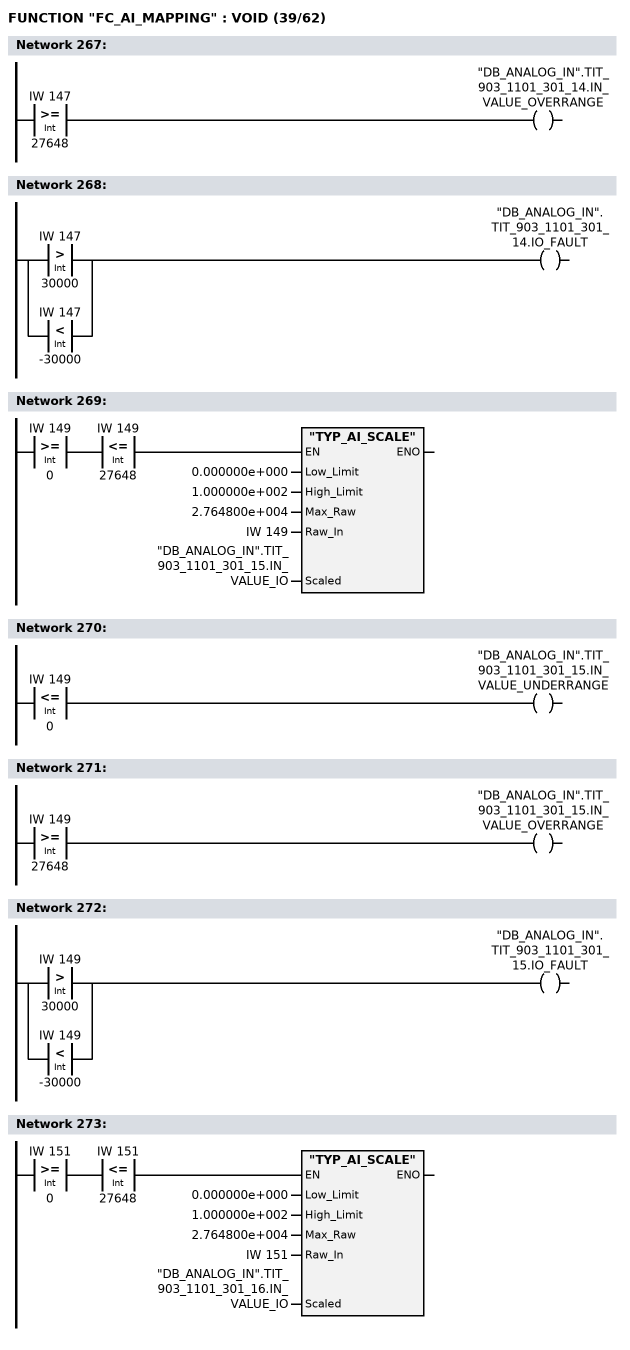

      L     IW      147;
      L     27648;
      >=I   ;
      =     "DB_ANALOG_IN".TIT_903_1101_301_14.IN_VALUE_OVERRANGE;
NETWORK
TITLE =

      O(    ;
      L     IW      147;
      L     30000;
      >I    ;
      )     ;
      O(    ;
      L     IW      147;
      L     -30000;
      <I    ;
      )     ;
      =     "DB_ANALOG_IN".TIT_903_1101_301_14.IO_FAULT;

NETWORK
TITLE =

      A(    ;
      L     IW      149;
      L     0;
      >=I   ;
      )     ;
      A(    ;
      L     IW      149;

      L     27648;
      <=I   ;
      )     ;
      JNB   _044;
      CALL "TYP_AI_SCALE" (
           Low_Limit                := 0.000000e+000,
           High_Limit               := 1.000000e+002,
           Max_Raw                  := 2.764800e+004,
           Raw_In                   := IW      149,
           Scaled                   := "DB_ANALOG_IN".TIT_903_1101_301_15.IN_VALUE_IO);
_044: NOP   0;
NETWORK
TITLE =

      L     IW      149;
      L     0;
      <=I   ;
      =     "DB_ANALOG_IN".TIT_903_1101_301_15.IN_VALUE_UNDERRANGE;
NETWORK
TITLE =

      L     IW      149;
      L     27648;
      >=I   ;
      =     "DB_ANALOG_IN".TIT_903_1101_301_15.IN_VALUE_OVERRANGE;
NETWORK
TITLE =

      O(    ;
      L     IW      149;
      L     30000;
      >I    ;
      )     ;
      O(    ;
      L     IW      149;
      L     -30000;
      <I    ;
      )     ;
      =     "DB_ANALOG_IN".TIT_903_1101_301_15.IO_FAULT;

NETWORK
TITLE =

      A(    ;
      L     IW      151;
      L     0;
      >=I   ;
      )     ;
      A(    ;
      L     IW      151;

      L     27648;
      <=I   ;
      )     ;
      JNB   _045;
      CALL "TYP_AI_SCALE" (
           Low_Limit                := 0.000000e+000,
           High_Limit               := 1.000000e+002,
           Max_Raw                  := 2.764800e+004,
           Raw_In                   := IW      151,
           Scaled                   := "DB_ANALOG_IN".TIT_903_1101_301_16.IN_VALUE_IO);
_045: NOP   0;
NETWORK
TITLE =
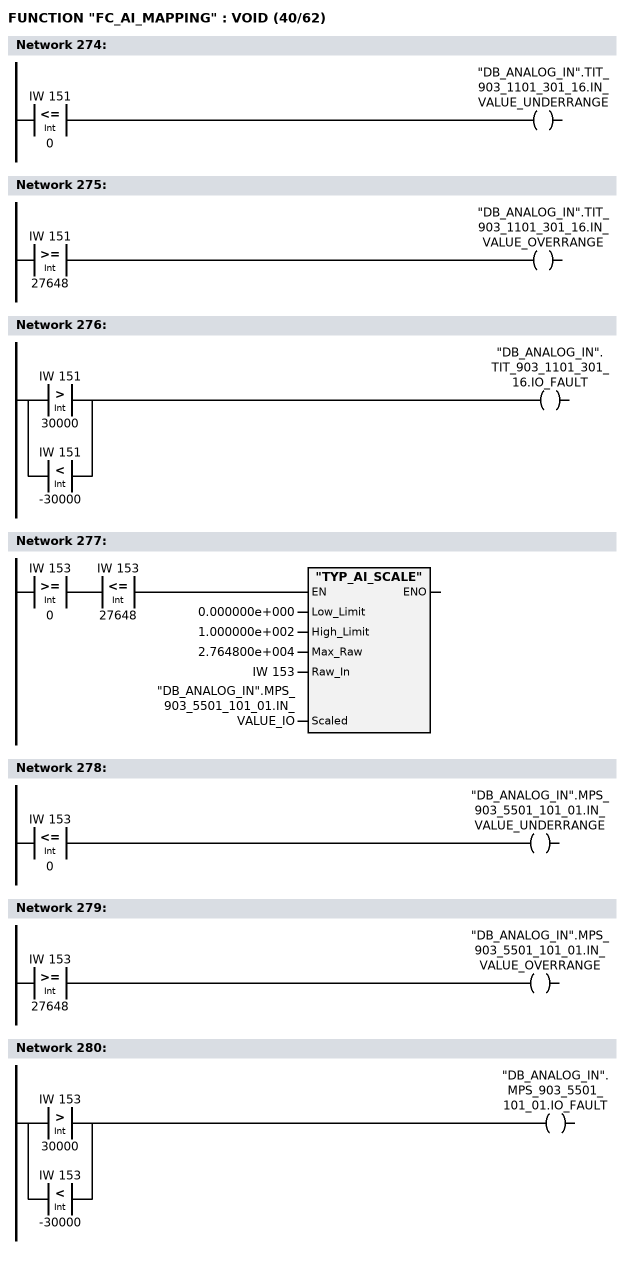

      L     IW      151;
      L     0;
      <=I   ;
      =     "DB_ANALOG_IN".TIT_903_1101_301_16.IN_VALUE_UNDERRANGE;
NETWORK
TITLE =

      L     IW      151;
      L     27648;
      >=I   ;
      =     "DB_ANALOG_IN".TIT_903_1101_301_16.IN_VALUE_OVERRANGE;
NETWORK
TITLE =

      O(    ;
      L     IW      151;
      L     30000;
      >I    ;
      )     ;
      O(    ;
      L     IW      151;
      L     -30000;
      <I    ;
      )     ;
      =     "DB_ANALOG_IN".TIT_903_1101_301_16.IO_FAULT;

NETWORK
TITLE =

      A(    ;
      L     IW      153;
      L     0;
      >=I   ;
      )     ;
      A(    ;
      L     IW      153;

      L     27648;
      <=I   ;
      )     ;
      JNB   _046;
      CALL "TYP_AI_SCALE" (
           Low_Limit                := 0.000000e+000,
           High_Limit               := 1.000000e+002,
           Max_Raw                  := 2.764800e+004,
           Raw_In                   := IW      153,
           Scaled                   := "DB_ANALOG_IN".MPS_903_5501_101_01.IN_VALUE_IO);
_046: NOP   0;
NETWORK
TITLE =

      L     IW      153;
      L     0;
      <=I   ;
      =     "DB_ANALOG_IN".MPS_903_5501_101_01.IN_VALUE_UNDERRANGE;
NETWORK
TITLE =

      L     IW      153;
      L     27648;
      >=I   ;
      =     "DB_ANALOG_IN".MPS_903_5501_101_01.IN_VALUE_OVERRANGE;
NETWORK
TITLE =

      O(    ;
      L     IW      153;
      L     30000;
      >I    ;
      )     ;
      O(    ;
      L     IW      153;
      L     -30000;
      <I    ;
      )     ;
      =     "DB_ANALOG_IN".MPS_903_5501_101_01.IO_FAULT;

NETWORK
TITLE =
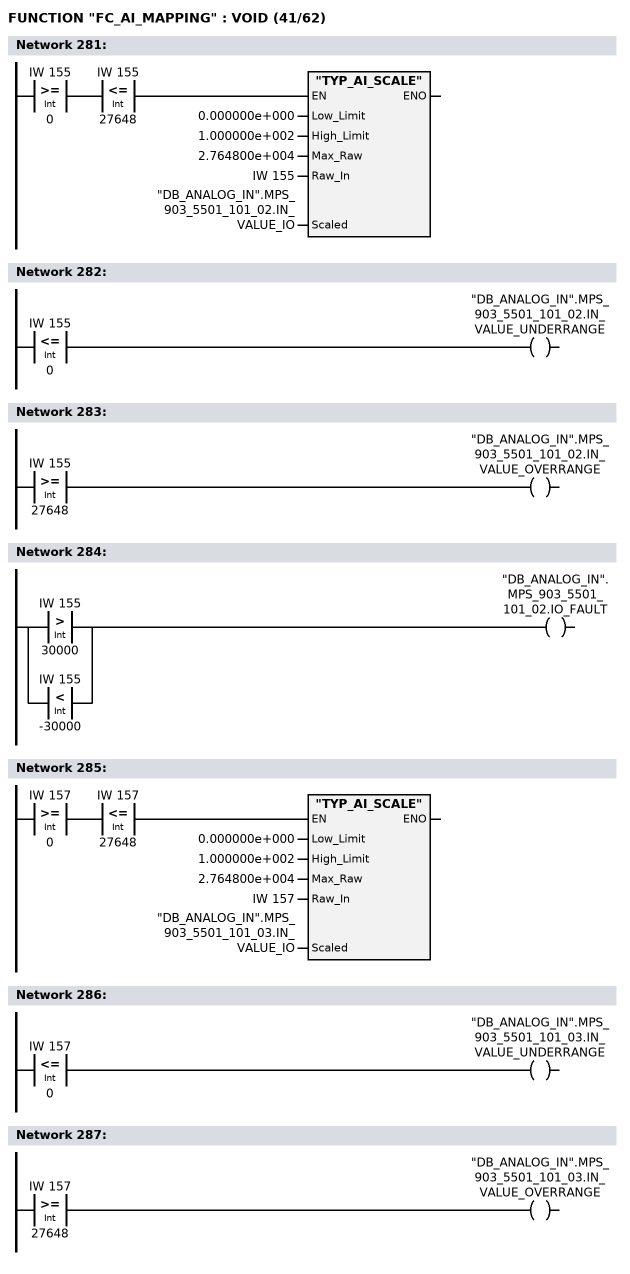

      A(    ;
      L     IW      155;
      L     0;
      >=I   ;
      )     ;
      A(    ;
      L     IW      155;

      L     27648;
      <=I   ;
      )     ;
      JNB   _047;
      CALL "TYP_AI_SCALE" (
           Low_Limit                := 0.000000e+000,
           High_Limit               := 1.000000e+002,
           Max_Raw                  := 2.764800e+004,
           Raw_In                   := IW      155,
           Scaled                   := "DB_ANALOG_IN".MPS_903_5501_101_02.IN_VALUE_IO);
_047: NOP   0;
NETWORK
TITLE =

      L     IW      155;
      L     0;
      <=I   ;
      =     "DB_ANALOG_IN".MPS_903_5501_101_02.IN_VALUE_UNDERRANGE;
NETWORK
TITLE =

      L     IW      155;
      L     27648;
      >=I   ;
      =     "DB_ANALOG_IN".MPS_903_5501_101_02.IN_VALUE_OVERRANGE;
NETWORK
TITLE =

      O(    ;
      L     IW      155;
      L     30000;
      >I    ;
      )     ;
      O(    ;
      L     IW      155;
      L     -30000;
      <I    ;
      )     ;
      =     "DB_ANALOG_IN".MPS_903_5501_101_02.IO_FAULT;

NETWORK
TITLE =

      A(    ;
      L     IW      157;
      L     0;
      >=I   ;
      )     ;
      A(    ;
      L     IW      157;

      L     27648;
      <=I   ;
      )     ;
      JNB   _048;
      CALL "TYP_AI_SCALE" (
           Low_Limit                := 0.000000e+000,
           High_Limit               := 1.000000e+002,
           Max_Raw                  := 2.764800e+004,
           Raw_In                   := IW      157,
           Scaled                   := "DB_ANALOG_IN".MPS_903_5501_101_03.IN_VALUE_IO);
_048: NOP   0;
NETWORK
TITLE =

      L     IW      157;
      L     0;
      <=I   ;
      =     "DB_ANALOG_IN".MPS_903_5501_101_03.IN_VALUE_UNDERRANGE;
NETWORK
TITLE =

      L     IW      157;
      L     27648;
      >=I   ;
      =     "DB_ANALOG_IN".MPS_903_5501_101_03.IN_VALUE_OVERRANGE;
NETWORK
TITLE =
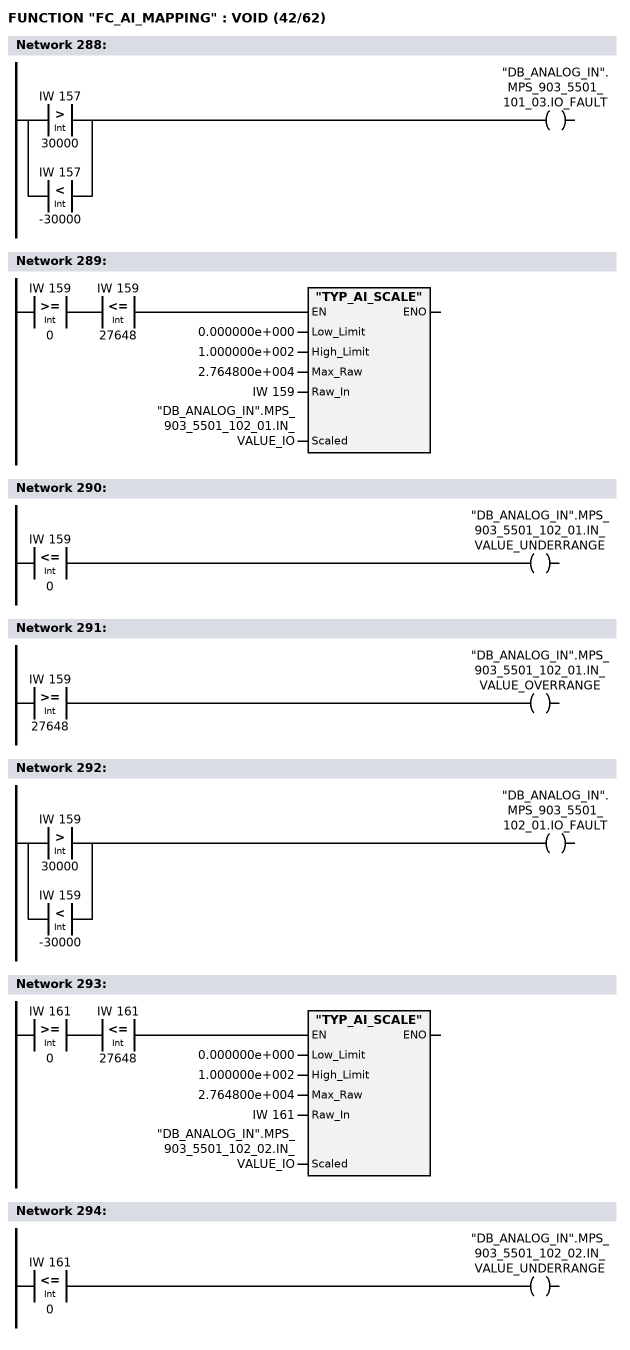

      O(    ;
      L     IW      157;
      L     30000;
      >I    ;
      )     ;
      O(    ;
      L     IW      157;
      L     -30000;
      <I    ;
      )     ;
      =     "DB_ANALOG_IN".MPS_903_5501_101_03.IO_FAULT;

NETWORK
TITLE =

      A(    ;
      L     IW      159;
      L     0;
      >=I   ;
      )     ;
      A(    ;
      L     IW      159;

      L     27648;
      <=I   ;
      )     ;
      JNB   _049;
      CALL "TYP_AI_SCALE" (
           Low_Limit                := 0.000000e+000,
           High_Limit               := 1.000000e+002,
           Max_Raw                  := 2.764800e+004,
           Raw_In                   := IW      159,
           Scaled                   := "DB_ANALOG_IN".MPS_903_5501_102_01.IN_VALUE_IO);
_049: NOP   0;
NETWORK
TITLE =

      L     IW      159;
      L     0;
      <=I   ;
      =     "DB_ANALOG_IN".MPS_903_5501_102_01.IN_VALUE_UNDERRANGE;
NETWORK
TITLE =

      L     IW      159;
      L     27648;
      >=I   ;
      =     "DB_ANALOG_IN".MPS_903_5501_102_01.IN_VALUE_OVERRANGE;
NETWORK
TITLE =

      O(    ;
      L     IW      159;
      L     30000;
      >I    ;
      )     ;
      O(    ;
      L     IW      159;
      L     -30000;
      <I    ;
      )     ;
      =     "DB_ANALOG_IN".MPS_903_5501_102_01.IO_FAULT;

NETWORK
TITLE =

      A(    ;
      L     IW      161;
      L     0;
      >=I   ;
      )     ;
      A(    ;
      L     IW      161;

      L     27648;
      <=I   ;
      )     ;
      JNB   _04a;
      CALL "TYP_AI_SCALE" (
           Low_Limit                := 0.000000e+000,
           High_Limit               := 1.000000e+002,
           Max_Raw                  := 2.764800e+004,
           Raw_In                   := IW      161,
           Scaled                   := "DB_ANALOG_IN".MPS_903_5501_102_02.IN_VALUE_IO);
_04a: NOP   0;
NETWORK
TITLE =

      L     IW      161;
      L     0;
      <=I   ;
      =     "DB_ANALOG_IN".MPS_903_5501_102_02.IN_VALUE_UNDERRANGE;
NETWORK
TITLE =
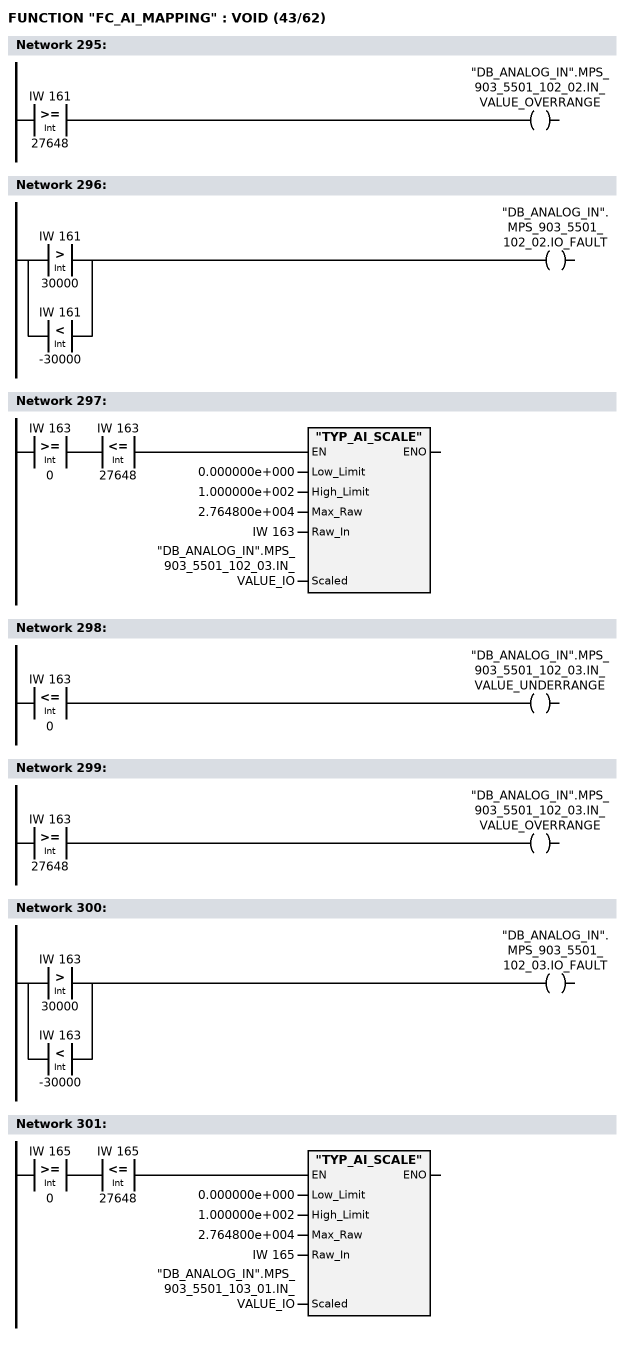

      L     IW      161;
      L     27648;
      >=I   ;
      =     "DB_ANALOG_IN".MPS_903_5501_102_02.IN_VALUE_OVERRANGE;
NETWORK
TITLE =

      O(    ;
      L     IW      161;
      L     30000;
      >I    ;
      )     ;
      O(    ;
      L     IW      161;
      L     -30000;
      <I    ;
      )     ;
      =     "DB_ANALOG_IN".MPS_903_5501_102_02.IO_FAULT;

NETWORK
TITLE =

      A(    ;
      L     IW      163;
      L     0;
      >=I   ;
      )     ;
      A(    ;
      L     IW      163;

      L     27648;
      <=I   ;
      )     ;
      JNB   _04b;
      CALL "TYP_AI_SCALE" (
           Low_Limit                := 0.000000e+000,
           High_Limit               := 1.000000e+002,
           Max_Raw                  := 2.764800e+004,
           Raw_In                   := IW      163,
           Scaled                   := "DB_ANALOG_IN".MPS_903_5501_102_03.IN_VALUE_IO);
_04b: NOP   0;
NETWORK
TITLE =

      L     IW      163;
      L     0;
      <=I   ;
      =     "DB_ANALOG_IN".MPS_903_5501_102_03.IN_VALUE_UNDERRANGE;
NETWORK
TITLE =

      L     IW      163;
      L     27648;
      >=I   ;
      =     "DB_ANALOG_IN".MPS_903_5501_102_03.IN_VALUE_OVERRANGE;
NETWORK
TITLE =

      O(    ;
      L     IW      163;
      L     30000;
      >I    ;
      )     ;
      O(    ;
      L     IW      163;
      L     -30000;
      <I    ;
      )     ;
      =     "DB_ANALOG_IN".MPS_903_5501_102_03.IO_FAULT;

NETWORK
TITLE =

      A(    ;
      L     IW      165;
      L     0;
      >=I   ;
      )     ;
      A(    ;
      L     IW      165;

      L     27648;
      <=I   ;
      )     ;
      JNB   _04c;
      CALL "TYP_AI_SCALE" (
           Low_Limit                := 0.000000e+000,
           High_Limit               := 1.000000e+002,
           Max_Raw                  := 2.764800e+004,
           Raw_In                   := IW      165,
           Scaled                   := "DB_ANALOG_IN".MPS_903_5501_103_01.IN_VALUE_IO);
_04c: NOP   0;
NETWORK
TITLE =
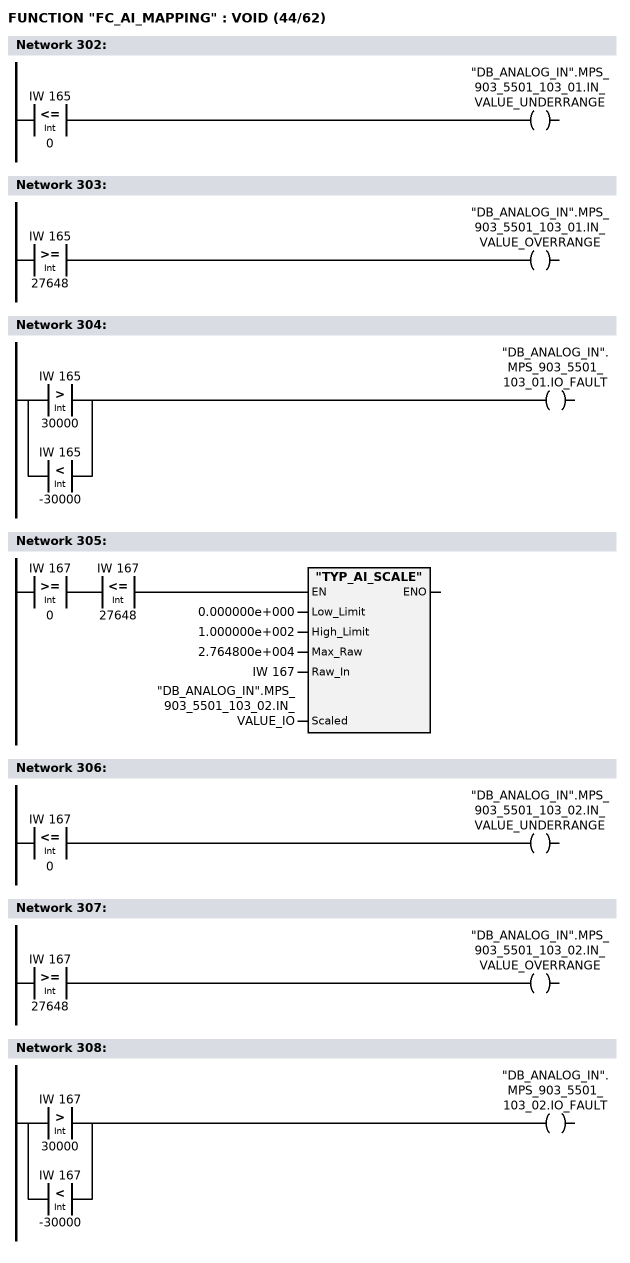

      L     IW      165;
      L     0;
      <=I   ;
      =     "DB_ANALOG_IN".MPS_903_5501_103_01.IN_VALUE_UNDERRANGE;
NETWORK
TITLE =

      L     IW      165;
      L     27648;
      >=I   ;
      =     "DB_ANALOG_IN".MPS_903_5501_103_01.IN_VALUE_OVERRANGE;
NETWORK
TITLE =

      O(    ;
      L     IW      165;
      L     30000;
      >I    ;
      )     ;
      O(    ;
      L     IW      165;
      L     -30000;
      <I    ;
      )     ;
      =     "DB_ANALOG_IN".MPS_903_5501_103_01.IO_FAULT;

NETWORK
TITLE =

      A(    ;
      L     IW      167;
      L     0;
      >=I   ;
      )     ;
      A(    ;
      L     IW      167;

      L     27648;
      <=I   ;
      )     ;
      JNB   _04d;
      CALL "TYP_AI_SCALE" (
           Low_Limit                := 0.000000e+000,
           High_Limit               := 1.000000e+002,
           Max_Raw                  := 2.764800e+004,
           Raw_In                   := IW      167,
           Scaled                   := "DB_ANALOG_IN".MPS_903_5501_103_02.IN_VALUE_IO);
_04d: NOP   0;
NETWORK
TITLE =

      L     IW      167;
      L     0;
      <=I   ;
      =     "DB_ANALOG_IN".MPS_903_5501_103_02.IN_VALUE_UNDERRANGE;
NETWORK
TITLE =

      L     IW      167;
      L     27648;
      >=I   ;
      =     "DB_ANALOG_IN".MPS_903_5501_103_02.IN_VALUE_OVERRANGE;
NETWORK
TITLE =

      O(    ;
      L     IW      167;
      L     30000;
      >I    ;
      )     ;
      O(    ;
      L     IW      167;
      L     -30000;
      <I    ;
      )     ;
      =     "DB_ANALOG_IN".MPS_903_5501_103_02.IO_FAULT;

NETWORK
TITLE =
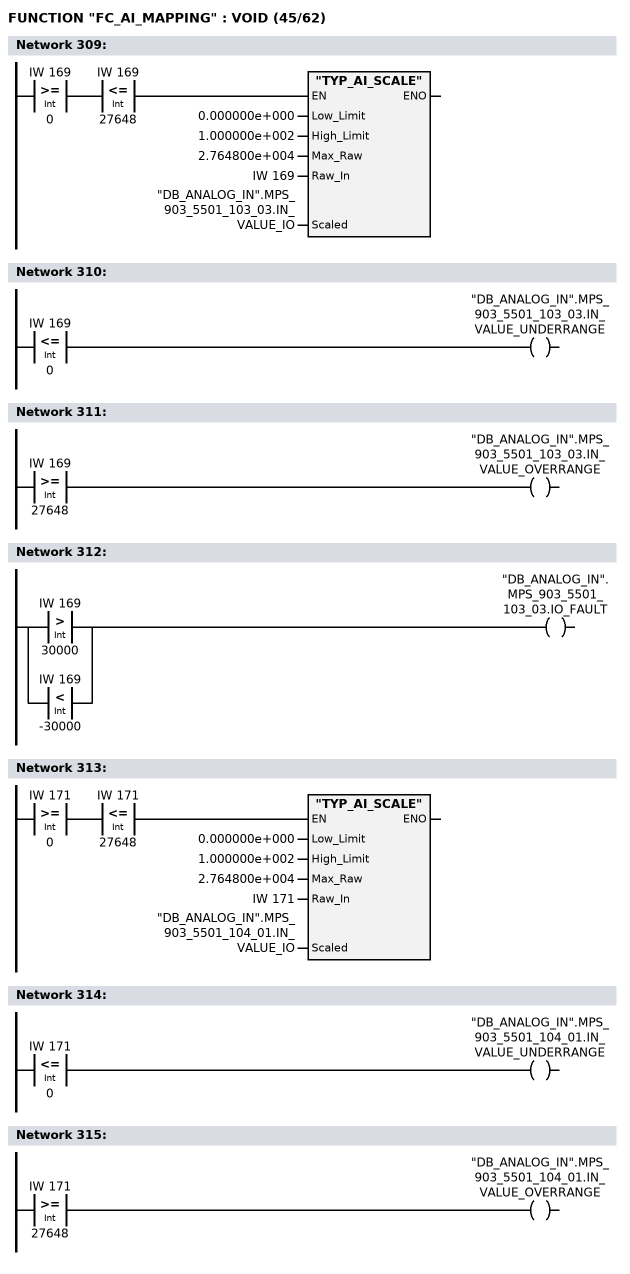

      A(    ;
      L     IW      169;
      L     0;
      >=I   ;
      )     ;
      A(    ;
      L     IW      169;

      L     27648;
      <=I   ;
      )     ;
      JNB   _04e;
      CALL "TYP_AI_SCALE" (
           Low_Limit                := 0.000000e+000,
           High_Limit               := 1.000000e+002,
           Max_Raw                  := 2.764800e+004,
           Raw_In                   := IW      169,
           Scaled                   := "DB_ANALOG_IN".MPS_903_5501_103_03.IN_VALUE_IO);
_04e: NOP   0;
NETWORK
TITLE =

      L     IW      169;
      L     0;
      <=I   ;
      =     "DB_ANALOG_IN".MPS_903_5501_103_03.IN_VALUE_UNDERRANGE;
NETWORK
TITLE =

      L     IW      169;
      L     27648;
      >=I   ;
      =     "DB_ANALOG_IN".MPS_903_5501_103_03.IN_VALUE_OVERRANGE;
NETWORK
TITLE =

      O(    ;
      L     IW      169;
      L     30000;
      >I    ;
      )     ;
      O(    ;
      L     IW      169;
      L     -30000;
      <I    ;
      )     ;
      =     "DB_ANALOG_IN".MPS_903_5501_103_03.IO_FAULT;

NETWORK
TITLE =

      A(    ;
      L     IW      171;
      L     0;
      >=I   ;
      )     ;
      A(    ;
      L     IW      171;

      L     27648;
      <=I   ;
      )     ;
      JNB   _04f;
      CALL "TYP_AI_SCALE" (
           Low_Limit                := 0.000000e+000,
           High_Limit               := 1.000000e+002,
           Max_Raw                  := 2.764800e+004,
           Raw_In                   := IW      171,
           Scaled                   := "DB_ANALOG_IN".MPS_903_5501_104_01.IN_VALUE_IO);
_04f: NOP   0;
NETWORK
TITLE =

      L     IW      171;
      L     0;
      <=I   ;
      =     "DB_ANALOG_IN".MPS_903_5501_104_01.IN_VALUE_UNDERRANGE;
NETWORK
TITLE =

      L     IW      171;
      L     27648;
      >=I   ;
      =     "DB_ANALOG_IN".MPS_903_5501_104_01.IN_VALUE_OVERRANGE;
NETWORK
TITLE =
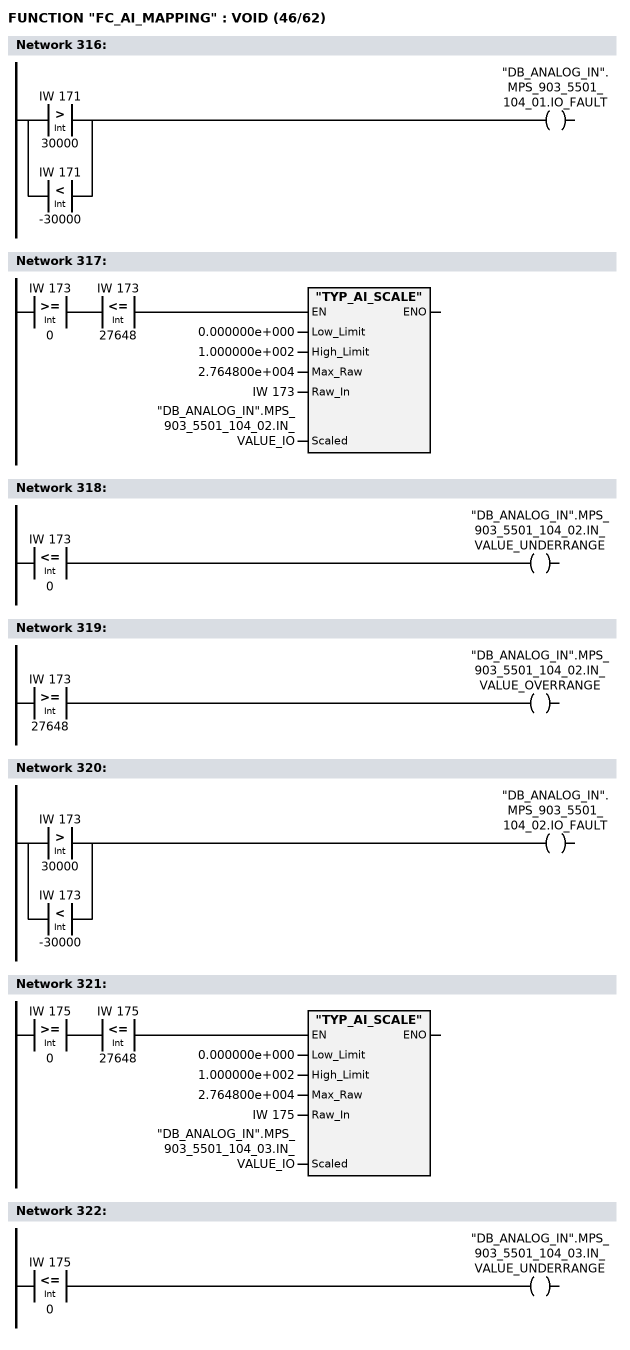

      O(    ;
      L     IW      171;
      L     30000;
      >I    ;
      )     ;
      O(    ;
      L     IW      171;
      L     -30000;
      <I    ;
      )     ;
      =     "DB_ANALOG_IN".MPS_903_5501_104_01.IO_FAULT;

NETWORK
TITLE =

      A(    ;
      L     IW      173;
      L     0;
      >=I   ;
      )     ;
      A(    ;
      L     IW      173;

      L     27648;
      <=I   ;
      )     ;
      JNB   _050;
      CALL "TYP_AI_SCALE" (
           Low_Limit                := 0.000000e+000,
           High_Limit               := 1.000000e+002,
           Max_Raw                  := 2.764800e+004,
           Raw_In                   := IW      173,
           Scaled                   := "DB_ANALOG_IN".MPS_903_5501_104_02.IN_VALUE_IO);
_050: NOP   0;
NETWORK
TITLE =

      L     IW      173;
      L     0;
      <=I   ;
      =     "DB_ANALOG_IN".MPS_903_5501_104_02.IN_VALUE_UNDERRANGE;
NETWORK
TITLE =

      L     IW      173;
      L     27648;
      >=I   ;
      =     "DB_ANALOG_IN".MPS_903_5501_104_02.IN_VALUE_OVERRANGE;
NETWORK
TITLE =

      O(    ;
      L     IW      173;
      L     30000;
      >I    ;
      )     ;
      O(    ;
      L     IW      173;
      L     -30000;
      <I    ;
      )     ;
      =     "DB_ANALOG_IN".MPS_903_5501_104_02.IO_FAULT;

NETWORK
TITLE =

      A(    ;
      L     IW      175;
      L     0;
      >=I   ;
      )     ;
      A(    ;
      L     IW      175;

      L     27648;
      <=I   ;
      )     ;
      JNB   _051;
      CALL "TYP_AI_SCALE" (
           Low_Limit                := 0.000000e+000,
           High_Limit               := 1.000000e+002,
           Max_Raw                  := 2.764800e+004,
           Raw_In                   := IW      175,
           Scaled                   := "DB_ANALOG_IN".MPS_903_5501_104_03.IN_VALUE_IO);
_051: NOP   0;
NETWORK
TITLE =

      L     IW      175;
      L     0;
      <=I   ;
      =     "DB_ANALOG_IN".MPS_903_5501_104_03.IN_VALUE_UNDERRANGE;
NETWORK
TITLE =
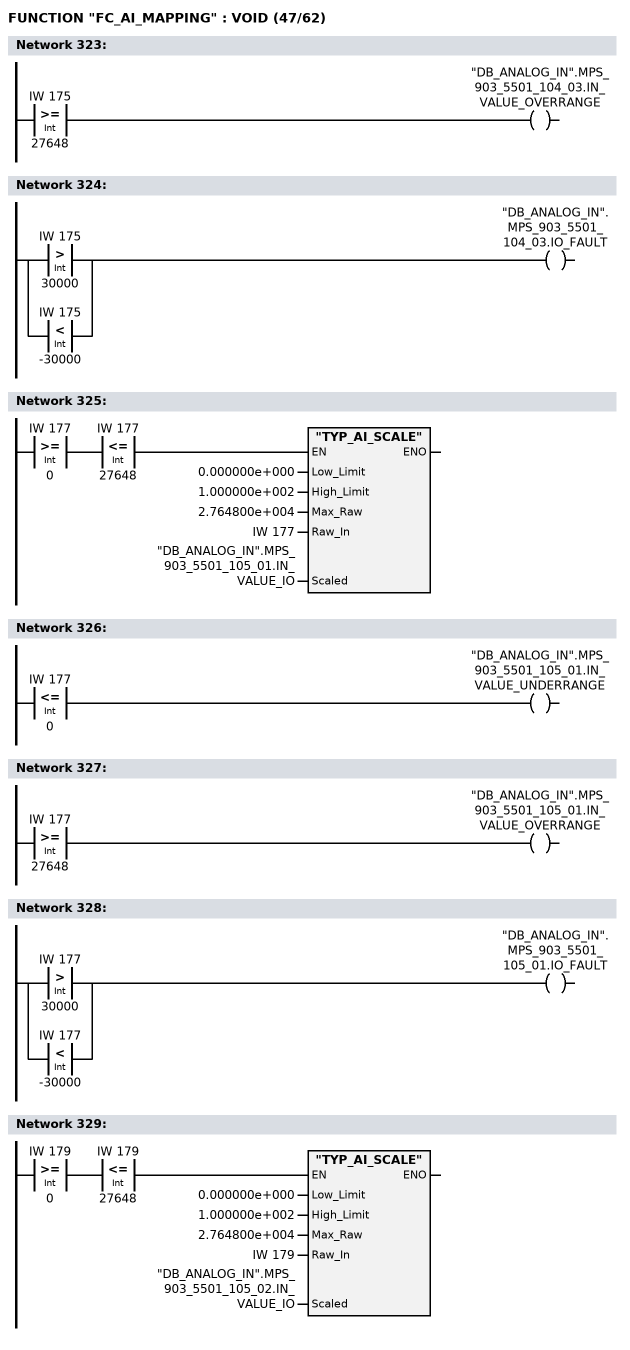

      L     IW      175;
      L     27648;
      >=I   ;
      =     "DB_ANALOG_IN".MPS_903_5501_104_03.IN_VALUE_OVERRANGE;
NETWORK
TITLE =

      O(    ;
      L     IW      175;
      L     30000;
      >I    ;
      )     ;
      O(    ;
      L     IW      175;
      L     -30000;
      <I    ;
      )     ;
      =     "DB_ANALOG_IN".MPS_903_5501_104_03.IO_FAULT;

NETWORK
TITLE =

      A(    ;
      L     IW      177;
      L     0;
      >=I   ;
      )     ;
      A(    ;
      L     IW      177;

      L     27648;
      <=I   ;
      )     ;
      JNB   _052;
      CALL "TYP_AI_SCALE" (
           Low_Limit                := 0.000000e+000,
           High_Limit               := 1.000000e+002,
           Max_Raw                  := 2.764800e+004,
           Raw_In                   := IW      177,
           Scaled                   := "DB_ANALOG_IN".MPS_903_5501_105_01.IN_VALUE_IO);
_052: NOP   0;
NETWORK
TITLE =

      L     IW      177;
      L     0;
      <=I   ;
      =     "DB_ANALOG_IN".MPS_903_5501_105_01.IN_VALUE_UNDERRANGE;
NETWORK
TITLE =

      L     IW      177;
      L     27648;
      >=I   ;
      =     "DB_ANALOG_IN".MPS_903_5501_105_01.IN_VALUE_OVERRANGE;
NETWORK
TITLE =

      O(    ;
      L     IW      177;
      L     30000;
      >I    ;
      )     ;
      O(    ;
      L     IW      177;
      L     -30000;
      <I    ;
      )     ;
      =     "DB_ANALOG_IN".MPS_903_5501_105_01.IO_FAULT;

NETWORK
TITLE =

      A(    ;
      L     IW      179;
      L     0;
      >=I   ;
      )     ;
      A(    ;
      L     IW      179;

      L     27648;
      <=I   ;
      )     ;
      JNB   _053;
      CALL "TYP_AI_SCALE" (
           Low_Limit                := 0.000000e+000,
           High_Limit               := 1.000000e+002,
           Max_Raw                  := 2.764800e+004,
           Raw_In                   := IW      179,
           Scaled                   := "DB_ANALOG_IN".MPS_903_5501_105_02.IN_VALUE_IO);
_053: NOP   0;
NETWORK
TITLE =
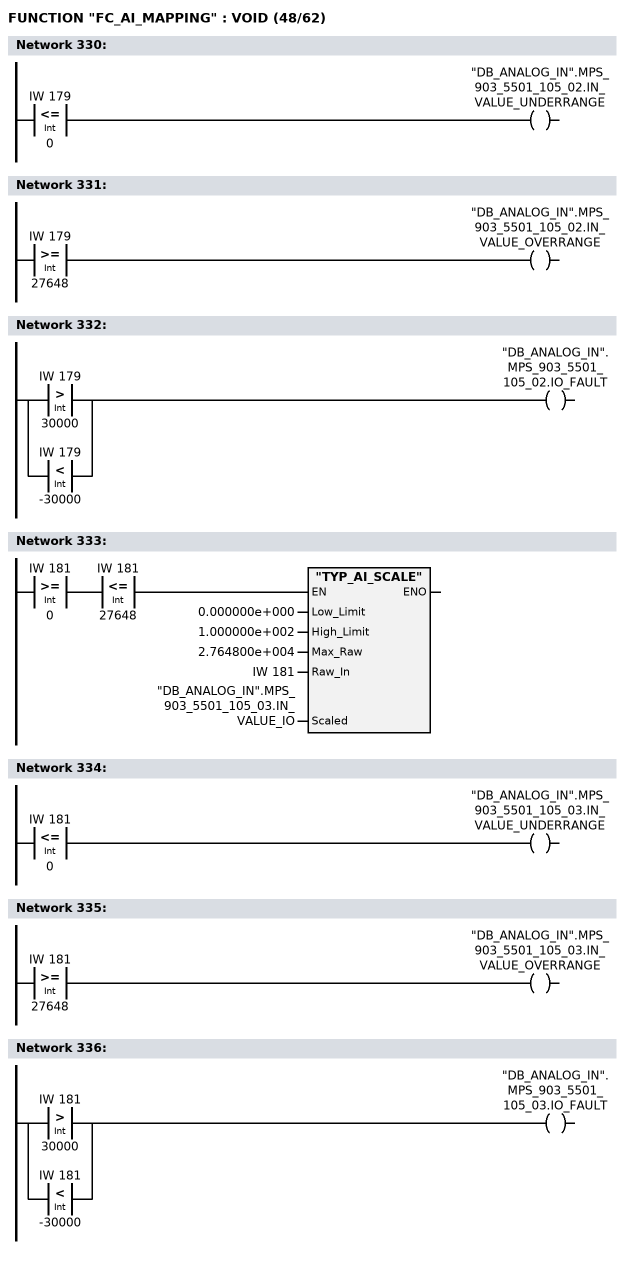

      L     IW      179;
      L     0;
      <=I   ;
      =     "DB_ANALOG_IN".MPS_903_5501_105_02.IN_VALUE_UNDERRANGE;
NETWORK
TITLE =

      L     IW      179;
      L     27648;
      >=I   ;
      =     "DB_ANALOG_IN".MPS_903_5501_105_02.IN_VALUE_OVERRANGE;
NETWORK
TITLE =

      O(    ;
      L     IW      179;
      L     30000;
      >I    ;
      )     ;
      O(    ;
      L     IW      179;
      L     -30000;
      <I    ;
      )     ;
      =     "DB_ANALOG_IN".MPS_903_5501_105_02.IO_FAULT;

NETWORK
TITLE =

      A(    ;
      L     IW      181;
      L     0;
      >=I   ;
      )     ;
      A(    ;
      L     IW      181;

      L     27648;
      <=I   ;
      )     ;
      JNB   _054;
      CALL "TYP_AI_SCALE" (
           Low_Limit                := 0.000000e+000,
           High_Limit               := 1.000000e+002,
           Max_Raw                  := 2.764800e+004,
           Raw_In                   := IW      181,
           Scaled                   := "DB_ANALOG_IN".MPS_903_5501_105_03.IN_VALUE_IO);
_054: NOP   0;
NETWORK
TITLE =

      L     IW      181;
      L     0;
      <=I   ;
      =     "DB_ANALOG_IN".MPS_903_5501_105_03.IN_VALUE_UNDERRANGE;
NETWORK
TITLE =

      L     IW      181;
      L     27648;
      >=I   ;
      =     "DB_ANALOG_IN".MPS_903_5501_105_03.IN_VALUE_OVERRANGE;
NETWORK
TITLE =

      O(    ;
      L     IW      181;
      L     30000;
      >I    ;
      )     ;
      O(    ;
      L     IW      181;
      L     -30000;
      <I    ;
      )     ;
      =     "DB_ANALOG_IN".MPS_903_5501_105_03.IO_FAULT;

NETWORK
TITLE =
